  MoveL 7398 to (239.35, 44.42, 106.87) mm, rotated rx -180 ry 0 rz 180 deg; joints [-29.24, 54.738, -85.05, 32.961, 116.129, 15.937]
  Call Extruder(207.44470)
  MoveL 7399 to (239.44, 44.66, 106.87) mm, rotated rx 180 ry 0 rz 180 deg; joints [-29.343, 54.76, -85.048, 33.066, 116.082, 15.973]
  MoveL 7400 to (239.44, 44.66, 106.87) mm, rotated rx 180 ry 0 rz 180 deg; joints [-29.343, 54.76, -85.048, 33.066, 116.082, 15.973]
  Call Extruder(207.55794)
  MoveL 7401 to (239.5, 44.85, 106.87) mm, rotated rx 180 ry 0 rz 180 deg; joints [-29.428, 54.775, -85.047, 33.152, 116.044, 16.002]
  MoveL 7402 to (239.5, 44.85, 106.87) mm, rotated rx 180 ry 0 rz 180 deg; joints [-29.428, 54.775, -85.047, 33.152, 116.044, 16.002]
  Call Extruder(207.67073)
  MoveL 7403 to (239.56, 45.03, 106.87) mm, rotated rx 180 ry 0 rz 180 deg; joints [-29.512, 54.791, -85.047, 33.237, 116.007, 16.031]
  MoveL 7404 to (239.56, 45.03, 106.87) mm, rotated rx 180 ry 0 rz 180 deg; joints [-29.512, 54.791, -85.047, 33.237, 116.007, 16.031]
  Call Extruder(207.78308)
  MoveL 7405 to (239.62, 45.22, 106.87) mm, rotated rx -180 ry 0 rz 180 deg; joints [-29.596, 54.807, -85.046, 33.322, 115.97, 16.061]
  MoveL 7406 to (239.62, 45.22, 106.87) mm, rotated rx -180 ry 0 rz 180 deg; joints [-29.596, 54.807, -85.046, 33.322, 115.97, 16.061]
  Call Extruder(207.89498)
  MoveL 7407 to (239.68, 45.41, 106.87) mm, rotated rx 180 ry 0 rz 180 deg; joints [-29.679, 54.822, -85.045, 33.407, 115.933, 16.089]
  MoveL 7408 to (239.68, 45.41, 106.87) mm, rotated rx 180 ry 0 rz 180 deg; joints [-29.679, 54.822, -85.045, 33.407, 115.933, 16.089]
  Call Extruder(208.01638)
  MoveL 7409 to (239.75, 45.62, 106.87) mm, rotated rx -180 ry 0 rz 180 deg; joints [-29.77, 54.839, -85.044, 33.5, 115.893, 16.121]
  MoveL 7410 to (239.75, 45.62, 106.87) mm, rotated rx -180 ry 0 rz 180 deg; joints [-29.77, 54.839, -85.044, 33.5, 115.893, 16.121]
  Call Extruder(208.14717)
  MoveL 7411 to (239.82, 45.84, 106.87) mm, rotated rx 180 ry 0 rz -180 deg; joints [-29.871, 54.858, -85.043, 33.601, 115.849, 16.156]
  MoveL 7412 to (239.82, 45.84, 106.87) mm, rotated rx 180 ry 0 rz -180 deg; joints [-29.871, 54.858, -85.043, 33.601, 115.849, 16.156]
  Call Extruder(208.27740)
  MoveL 7413 to (239.88, 46.06, 106.87) mm, rotated rx -180 ry 0 rz 180 deg; joints [-29.97, 54.876, -85.041, 33.702, 115.805, 16.19]
  MoveL 7414 to (239.88, 46.06, 106.87) mm, rotated rx -180 ry 0 rz 180 deg; joints [-29.97, 54.876, -85.041, 33.702, 115.805, 16.19]
  Call Extruder(208.40706)
  MoveL 7415 to (239.95, 46.29, 106.87) mm, rotated rx -180 ry 0 rz 180 deg; joints [-30.069, 54.894, -85.04, 33.803, 115.761, 16.224]
  MoveL 7416 to (239.95, 46.29, 106.87) mm, rotated rx -180 ry 0 rz 180 deg; joints [-30.069, 54.894, -85.04, 33.803, 115.761, 16.224]
  Call Extruder(208.53615)
  MoveL 7417 to (240.02, 46.51, 106.87) mm, rotated rx -180 ry 0 rz 180 deg; joints [-30.168, 54.913, -85.039, 33.903, 115.717, 16.258]
  MoveL 7418 to (240.02, 46.51, 106.87) mm, rotated rx -180 ry 0 rz 180 deg; joints [-30.168, 54.913, -85.039, 33.903, 115.717, 16.258]
  Call Extruder(208.65121)
  MoveL 7419 to (240.06, 46.72, 106.87) mm, rotated rx 180 ry 0 rz 180 deg; joints [-30.263, 54.928, -85.038, 34, 115.677, 16.292]
  MoveL 7420 to (240.06, 46.72, 106.87) mm, rotated rx 180 ry 0 rz 180 deg; joints [-30.263, 54.928, -85.038, 34, 115.677, 16.292]
  Call Extruder(208.76581)
  MoveL 7421 to (240.11, 46.92, 106.87) mm, rotated rx -180 ry 0 rz 180 deg; joints [-30.358, 54.943, -85.037, 34.097, 115.637, 16.326]
  MoveL 7422 to (240.11, 46.92, 106.87) mm, rotated rx -180 ry 0 rz 180 deg; joints [-30.358, 54.943, -85.037, 34.097, 115.637, 16.326]
  Call Extruder(208.87996)
  MoveL 7423 to (240.15, 47.12, 106.87) mm, rotated rx -180 ry 0 rz 180 deg; joints [-30.453, 54.958, -85.036, 34.193, 115.597, 16.359]
  MoveL 7424 to (240.15, 47.12, 106.87) mm, rotated rx -180 ry 0 rz 180 deg; joints [-30.453, 54.958, -85.036, 34.193, 115.597, 16.359]
  Call Extruder(208.99365)
  MoveL 7425 to (240.2, 47.33, 106.87) mm, rotated rx 180 ry 0 rz 180 deg; joints [-30.548, 54.973, -85.035, 34.29, 115.557, 16.393]
  MoveL 7426 to (240.2, 47.33, 106.87) mm, rotated rx 180 ry 0 rz 180 deg; joints [-30.548, 54.973, -85.035, 34.29, 115.557, 16.393]
  Call Extruder(209.11906)
  MoveL 7427 to (240.24, 47.55, 106.87) mm, rotated rx -180 ry 0 rz 180 deg; joints [-30.653, 54.99, -85.034, 34.396, 115.513, 16.43]
  MoveL 7428 to (240.24, 47.55, 106.87) mm, rotated rx -180 ry 0 rz 180 deg; joints [-30.653, 54.99, -85.034, 34.396, 115.513, 16.43]
  Call Extruder(209.25604)
  MoveL 7429 to (240.29, 47.8, 106.87) mm, rotated rx 180 ry 0 rz -180 deg; joints [-30.768, 55.008, -85.033, 34.514, 115.464, 16.47]
  MoveL 7430 to (240.29, 47.8, 106.87) mm, rotated rx 180 ry 0 rz -180 deg; joints [-30.768, 55.008, -85.033, 34.514, 115.464, 16.47]
  Call Extruder(209.39241)
  MoveL 7431 to (240.34, 48.05, 106.87) mm, rotated rx -180 ry 0 rz 180 deg; joints [-30.884, 55.026, -85.032, 34.632, 115.415, 16.511]
  MoveL 7432 to (240.34, 48.05, 106.87) mm, rotated rx -180 ry 0 rz 180 deg; joints [-30.884, 55.026, -85.032, 34.632, 115.415, 16.511]
  Call Extruder(209.52817)
  MoveL 7433 to (240.39, 48.3, 106.87) mm, rotated rx -180 ry 0 rz 180 deg; joints [-30.999, 55.045, -85.031, 34.749, 115.366, 16.551]
  MoveL 7434 to (240.39, 48.3, 106.87) mm, rotated rx -180 ry 0 rz 180 deg; joints [-30.999, 55.045, -85.031, 34.749, 115.366, 16.551]
  Call Extruder(209.66331)
  MoveL 7435 to (240.44, 48.55, 106.87) mm, rotated rx 180 ry 0 rz 180 deg; joints [-31.114, 55.063, -85.029, 34.865, 115.318, 16.591]
  MoveL 7436 to (240.44, 48.55, 106.87) mm, rotated rx 180 ry 0 rz 180 deg; joints [-31.114, 55.063, -85.029, 34.865, 115.318, 16.591]
  Call Extruder(209.79785)
  MoveL 7437 to (240.49, 48.8, 106.87) mm, rotated rx -180 ry 0 rz 180 deg; joints [-31.228, 55.081, -85.028, 34.981, 115.269, 16.63]
  MoveL 7438 to (240.49, 48.8, 106.87) mm, rotated rx -180 ry 0 rz 180 deg; joints [-31.228, 55.081, -85.028, 34.981, 115.269, 16.63]
  Call Extruder(209.93178)
  MoveL 7439 to (240.54, 49.05, 106.87) mm, rotated rx -180 ry 0 rz 180 deg; joints [-31.342, 55.1, -85.027, 35.096, 115.22, 16.669]
  MoveL 7440 to (240.54, 49.05, 106.87) mm, rotated rx -180 ry 0 rz 180 deg; joints [-31.342, 55.1, -85.027, 35.096, 115.22, 16.669]
  Call Extruder(210.07964)
  MoveL 7441 to (240.59, 49.33, 106.87) mm, rotated rx -180 ry 0 rz 180 deg; joints [-31.47, 55.12, -85.026, 35.226, 115.166, 16.713]
  MoveL 7442 to (240.59, 49.33, 106.87) mm, rotated rx -180 ry 0 rz 180 deg; joints [-31.47, 55.12, -85.026, 35.226, 115.166, 16.713]
  Call Extruder(210.24139)
  MoveL 7443 to (240.64, 49.63, 106.87) mm, rotated rx -180 ry 0 rz 180 deg; joints [-31.612, 55.141, -85.024, 35.37, 115.106, 16.762]
  MoveL 7444 to (240.64, 49.63, 106.87) mm, rotated rx -180 ry 0 rz 180 deg; joints [-31.612, 55.141, -85.024, 35.37, 115.106, 16.762]
  Call Extruder(210.40241)
  MoveL 7445 to (240.69, 49.94, 106.87) mm, rotated rx -180 ry 0 rz 180 deg; joints [-31.755, 55.163, -85.023, 35.514, 115.046, 16.811]
  MoveL 7446 to (240.69, 49.94, 106.87) mm, rotated rx -180 ry 0 rz 180 deg; joints [-31.755, 55.163, -85.023, 35.514, 115.046, 16.811]
  Call Extruder(210.56270)
  MoveL 7447 to (240.74, 50.24, 106.87) mm, rotated rx -180 ry 0 rz 180 deg; joints [-31.895, 55.184, -85.021, 35.657, 114.987, 16.859]
  MoveL 7448 to (240.74, 50.24, 106.87) mm, rotated rx -180 ry 0 rz 180 deg; joints [-31.895, 55.184, -85.021, 35.657, 114.987, 16.859]
  Call Extruder(210.72226)
  MoveL 7449 to (240.78, 50.55, 106.87) mm, rotated rx 180 ry 0 rz 180 deg; joints [-32.036, 55.206, -85.019, 35.799, 114.927, 16.907]
  MoveL 7450 to (240.78, 50.55, 106.87) mm, rotated rx 180 ry 0 rz 180 deg; joints [-32.036, 55.206, -85.019, 35.799, 114.927, 16.907]
  Call Extruder(210.88109)
  MoveL 7451 to (240.83, 50.86, 106.87) mm, rotated rx -180 ry 0 rz 180 deg; joints [-32.176, 55.228, -85.018, 35.941, 114.867, 16.954]
  MoveL 7452 to (240.83, 50.86, 106.87) mm, rotated rx -180 ry 0 rz 180 deg; joints [-32.176, 55.228, -85.018, 35.941, 114.867, 16.954]
  Call Extruder(211.05976)
  MoveL 7453 to (240.88, 51.2, 106.87) mm, rotated rx -180 ry 0 rz 180 deg; joints [-32.337, 55.252, -85.016, 36.103, 114.8, 17.009]
  MoveL 7454 to (240.88, 51.2, 106.87) mm, rotated rx -180 ry 0 rz 180 deg; joints [-32.337, 55.252, -85.016, 36.103, 114.8, 17.009]
  Call Extruder(211.25821)
  MoveL 7455 to (240.93, 51.59, 106.87) mm, rotated rx -180 ry 0 rz 180 deg; joints [-32.518, 55.278, -85.014, 36.285, 114.724, 17.07]
  MoveL 7456 to (240.93, 51.59, 106.87) mm, rotated rx -180 ry 0 rz 180 deg; joints [-32.518, 55.278, -85.014, 36.285, 114.724, 17.07]
  Call Extruder(211.45578)
  MoveL 7457 to (240.97, 51.98, 106.87) mm, rotated rx 180 ry 0 rz 180 deg; joints [-32.697, 55.304, -85.012, 36.467, 114.648, 17.131]
  MoveL 7458 to (240.97, 51.98, 106.87) mm, rotated rx 180 ry 0 rz 180 deg; joints [-32.697, 55.304, -85.012, 36.467, 114.648, 17.131]
  Call Extruder(211.65249)
  MoveL 7459 to (241.02, 52.37, 106.87) mm, rotated rx -180 ry 0 rz 180 deg; joints [-32.876, 55.331, -85.01, 36.647, 114.573, 17.19]
  MoveL 7460 to (241.02, 52.37, 106.87) mm, rotated rx -180 ry 0 rz 180 deg; joints [-32.876, 55.331, -85.01, 36.647, 114.573, 17.19]
  Call Extruder(211.84833)
  MoveL 7461 to (241.06, 52.75, 106.87) mm, rotated rx -180 ry 0 rz 180 deg; joints [-33.055, 55.357, -85.008, 36.826, 114.497, 17.249]
  MoveL 7462 to (241.06, 52.75, 106.87) mm, rotated rx -180 ry 0 rz 180 deg; joints [-33.055, 55.357, -85.008, 36.826, 114.497, 17.249]
  Call Extruder(212.14376)
  MoveL 7463 to (241.11, 53.34, 106.87) mm, rotated rx 180 ry 0 rz 180 deg; joints [-33.331, 55.396, -85.005, 37.105, 114.382, 17.342]
  MoveL 7464 to (241.11, 53.34, 106.87) mm, rotated rx 180 ry 0 rz 180 deg; joints [-33.331, 55.396, -85.005, 37.105, 114.382, 17.342]
  Call Extruder(212.43787)
  MoveL 7465 to (241.15, 53.93, 106.87) mm, rotated rx -180 ry 0 rz 180 deg; joints [-33.606, 55.434, -85.002, 37.381, 114.266, 17.433]
  MoveL 7466 to (241.15, 53.93, 106.87) mm, rotated rx -180 ry 0 rz 180 deg; joints [-33.606, 55.434, -85.002, 37.381, 114.266, 17.433]
  Call Extruder(212.73064)
  MoveL 7467 to (241.2, 54.52, 106.87) mm, rotated rx 180 ry 0 rz 180 deg; joints [-33.878, 55.473, -84.999, 37.655, 114.151, 17.521]
  MoveL 7468 to (241.2, 54.52, 106.87) mm, rotated rx 180 ry 0 rz 180 deg; joints [-33.878, 55.473, -84.999, 37.655, 114.151, 17.521]
  Call Extruder(213.30409)
  MoveL 7469 to (241.25, 55.68, 106.87) mm, rotated rx -180 ry 0 rz 180 deg; joints [-34.425, 55.546, -84.993, 38.203, 113.923, 17.7]
  MoveL 7470 to (241.25, 55.68, 106.87) mm, rotated rx -180 ry 0 rz 180 deg; joints [-34.425, 55.546, -84.993, 38.203, 113.923, 17.7]
  Call Extruder(214.01793)
  MoveL 7471 to (241.29, 57.14, 106.87) mm, rotated rx -180 ry 0 rz 180 deg; joints [-35.104, 55.637, -84.985, 38.883, 113.638, 17.918]
  Call Extruder(256.08281)
  MoveL 7472 to (241.29, 142.86, 106.87) mm, rotated rx 180 ry 0 rz 180 deg; joints [-60.361, 61.969, -83.576, 62.121, 100.493, 18.996]
  Call Extruder(256.51124)
  MoveL 7473 to (241.27, 143.74, 106.87) mm, rotated rx 180 ry 0 rz 180 deg; joints [-60.516, 62.035, -83.55, 62.255, 100.399, 18.94]
  MoveL 7474 to (241.27, 143.74, 106.87) mm, rotated rx 180 ry 0 rz 180 deg; joints [-60.516, 62.035, -83.55, 62.255, 100.399, 18.94]
  Call Extruder(257.08469)
  MoveL 7475 to (241.23, 144.9, 106.87) mm, rotated rx -180 ry 0 rz 180 deg; joints [-60.726, 62.123, -83.516, 62.438, 100.275, 18.867]
  MoveL 7476 to (241.23, 144.9, 106.87) mm, rotated rx -180 ry 0 rz 180 deg; joints [-60.726, 62.123, -83.516, 62.438, 100.275, 18.867]
  Call Extruder(257.51903)
  MoveL 7477 to (241.18, 145.77, 106.87) mm, rotated rx -180 ry 0 rz 180 deg; joints [-60.887, 62.188, -83.49, 62.578, 100.181, 18.812]
  MoveL 7478 to (241.18, 145.77, 106.87) mm, rotated rx -180 ry 0 rz 180 deg; joints [-60.887, 62.188, -83.49, 62.578, 100.181, 18.812]
  Call Extruder(257.81314)
  MoveL 7479 to (241.13, 146.36, 106.87) mm, rotated rx -180 ry 0 rz 180 deg; joints [-61, 62.231, -83.473, 62.676, 100.117, 18.777]
  MoveL 7480 to (241.13, 146.36, 106.87) mm, rotated rx -180 ry 0 rz 180 deg; joints [-61, 62.231, -83.473, 62.676, 100.117, 18.777]
  Call Extruder(258.10858)
  MoveL 7481 to (241.09, 146.95, 106.87) mm, rotated rx -180 ry 0 rz 180 deg; joints [-61.111, 62.275, -83.456, 62.774, 100.053, 18.741]
  MoveL 7482 to (241.09, 146.95, 106.87) mm, rotated rx -180 ry 0 rz 180 deg; joints [-61.111, 62.275, -83.456, 62.774, 100.053, 18.741]
  Call Extruder(258.35483)
  MoveL 7483 to (241.04, 147.44, 106.87) mm, rotated rx 180 ry 0 rz -180 deg; joints [-61.205, 62.31, -83.441, 62.857, 100, 18.712]
  MoveL 7484 to (241.04, 147.44, 106.87) mm, rotated rx 180 ry 0 rz -180 deg; joints [-61.205, 62.31, -83.441, 62.857, 100, 18.712]
  Call Extruder(258.55154)
  MoveL 7485 to (240.99, 147.83, 106.87) mm, rotated rx -180 ry 0 rz 180 deg; joints [-61.282, 62.338, -83.43, 62.925, 99.957, 18.689]
  MoveL 7486 to (240.99, 147.83, 106.87) mm, rotated rx -180 ry 0 rz 180 deg; joints [-61.282, 62.338, -83.43, 62.925, 99.957, 18.689]
  Call Extruder(258.74911)
  MoveL 7487 to (240.95, 148.22, 106.87) mm, rotated rx -180 ry 0 rz 180 deg; joints [-61.359, 62.366, -83.419, 62.992, 99.915, 18.667]
  MoveL 7488 to (240.95, 148.22, 106.87) mm, rotated rx -180 ry 0 rz 180 deg; joints [-61.359, 62.366, -83.419, 62.992, 99.915, 18.667]
  Call Extruder(258.94755)
  MoveL 7489 to (240.9, 148.6, 106.87) mm, rotated rx 180 ry 0 rz -180 deg; joints [-61.436, 62.393, -83.407, 63.06, 99.873, 18.644]
  MoveL 7490 to (240.9, 148.6, 106.87) mm, rotated rx 180 ry 0 rz -180 deg; joints [-61.436, 62.393, -83.407, 63.06, 99.873, 18.644]
  Call Extruder(259.14686)
  MoveL 7491 to (240.86, 148.99, 106.87) mm, rotated rx -180 ry 0 rz 180 deg; joints [-61.512, 62.421, -83.396, 63.127, 99.831, 18.621]
  MoveL 7492 to (240.86, 148.99, 106.87) mm, rotated rx -180 ry 0 rz 180 deg; joints [-61.512, 62.421, -83.396, 63.127, 99.831, 18.621]
  Call Extruder(259.30569)
  MoveL 7493 to (240.81, 149.3, 106.87) mm, rotated rx -180 ry 0 rz -180 deg; joints [-61.575, 62.443, -83.387, 63.184, 99.797, 18.604]
  MoveL 7494 to (240.81, 149.3, 106.87) mm, rotated rx -180 ry 0 rz -180 deg; joints [-61.575, 62.443, -83.387, 63.184, 99.797, 18.604]
  Call Extruder(259.46525)
  MoveL 7495 to (240.76, 149.6, 106.87) mm, rotated rx 180 ry 0 rz 180 deg; joints [-61.639, 62.464, -83.378, 63.24, 99.763, 18.587]
  MoveL 7496 to (240.76, 149.6, 106.87) mm, rotated rx 180 ry 0 rz 180 deg; joints [-61.639, 62.464, -83.378, 63.24, 99.763, 18.587]
  Call Extruder(259.62554)
  MoveL 7497 to (240.71, 149.91, 106.87) mm, rotated rx 180 ry 0 rz 180 deg; joints [-61.702, 62.485, -83.369, 63.296, 99.729, 18.57]
  MoveL 7498 to (240.71, 149.91, 106.87) mm, rotated rx 180 ry 0 rz 180 deg; joints [-61.702, 62.485, -83.369, 63.296, 99.729, 18.57]
  Call Extruder(259.78655)
  MoveL 7499 to (240.66, 150.21, 106.87) mm, rotated rx 180 ry 0 rz 180 deg; joints [-61.765, 62.507, -83.36, 63.352, 99.695, 18.552]
  MoveL 7500 to (240.66, 150.21, 106.87) mm, rotated rx 180 ry 0 rz 180 deg; joints [-61.765, 62.507, -83.36, 63.352, 99.695, 18.552]
  Call Extruder(259.94830)
  MoveL 7501 to (240.61, 150.52, 106.87) mm, rotated rx -180 ry 0 rz 180 deg; joints [-61.828, 62.528, -83.351, 63.408, 99.662, 18.535]
  MoveL 7502 to (240.61, 150.52, 106.87) mm, rotated rx -180 ry 0 rz 180 deg; joints [-61.828, 62.528, -83.351, 63.408, 99.662, 18.535]
  Call Extruder(260.11077)
  MoveL 7503 to (240.56, 150.83, 106.87) mm, rotated rx 180 ry 0 rz 180 deg; joints [-61.891, 62.55, -83.342, 63.464, 99.628, 18.518]
  MoveL 7504 to (240.56, 150.83, 106.87) mm, rotated rx 180 ry 0 rz 180 deg; joints [-61.891, 62.55, -83.342, 63.464, 99.628, 18.518]
  Call Extruder(260.24469)
  MoveL 7505 to (240.52, 151.07, 106.87) mm, rotated rx 180 ry 0 rz 180 deg; joints [-61.944, 62.567, -83.335, 63.512, 99.6, 18.504]
  MoveL 7506 to (240.52, 151.07, 106.87) mm, rotated rx 180 ry 0 rz 180 deg; joints [-61.944, 62.567, -83.335, 63.512, 99.6, 18.504]
  Call Extruder(260.37923)
  MoveL 7507 to (240.47, 151.32, 106.87) mm, rotated rx -180 ry 0 rz 180 deg; joints [-61.998, 62.584, -83.328, 63.56, 99.573, 18.491]
  MoveL 7508 to (240.47, 151.32, 106.87) mm, rotated rx -180 ry 0 rz 180 deg; joints [-61.998, 62.584, -83.328, 63.56, 99.573, 18.491]
  Call Extruder(260.51438)
  MoveL 7509 to (240.42, 151.57, 106.87) mm, rotated rx -180 ry 0 rz 180 deg; joints [-62.052, 62.601, -83.321, 63.608, 99.545, 18.477]
  MoveL 7510 to (240.42, 151.57, 106.87) mm, rotated rx -180 ry 0 rz 180 deg; joints [-62.052, 62.601, -83.321, 63.608, 99.545, 18.477]
  Call Extruder(260.65014)
  MoveL 7511 to (240.37, 151.82, 106.87) mm, rotated rx 180 ry 0 rz 180 deg; joints [-62.105, 62.618, -83.314, 63.656, 99.517, 18.464]
  MoveL 7512 to (240.37, 151.82, 106.87) mm, rotated rx 180 ry 0 rz 180 deg; joints [-62.105, 62.618, -83.314, 63.656, 99.517, 18.464]
  Call Extruder(260.78650)
  MoveL 7513 to (240.32, 152.07, 106.87) mm, rotated rx -180 ry 0 rz -180 deg; joints [-62.159, 62.635, -83.306, 63.704, 99.489, 18.45]
  MoveL 7514 to (240.32, 152.07, 106.87) mm, rotated rx -180 ry 0 rz -180 deg; joints [-62.159, 62.635, -83.306, 63.704, 99.489, 18.45]
  Call Extruder(260.92348)
  MoveL 7515 to (240.27, 152.32, 106.87) mm, rotated rx 180 ry 0 rz -180 deg; joints [-62.212, 62.652, -83.299, 63.751, 99.462, 18.437]
  MoveL 7516 to (240.27, 152.32, 106.87) mm, rotated rx 180 ry 0 rz -180 deg; joints [-62.212, 62.652, -83.299, 63.751, 99.462, 18.437]
  Call Extruder(261.06107)
  MoveL 7517 to (240.22, 152.57, 106.87) mm, rotated rx -180 ry 0 rz 180 deg; joints [-62.265, 62.669, -83.292, 63.799, 99.434, 18.423]
  MoveL 7518 to (240.22, 152.57, 106.87) mm, rotated rx -180 ry 0 rz 180 deg; joints [-62.265, 62.669, -83.292, 63.799, 99.434, 18.423]
  Call Extruder(261.17477)
  MoveL 7519 to (240.17, 152.77, 106.87) mm, rotated rx -180 ry 0 rz 180 deg; joints [-62.31, 62.683, -83.286, 63.839, 99.411, 18.412]
  MoveL 7520 to (240.17, 152.77, 106.87) mm, rotated rx -180 ry 0 rz 180 deg; joints [-62.31, 62.683, -83.286, 63.839, 99.411, 18.412]
  Call Extruder(261.28892)
  MoveL 7521 to (240.13, 152.98, 106.87) mm, rotated rx -180 ry 0 rz 180 deg; joints [-62.355, 62.696, -83.28, 63.879, 99.389, 18.401]
  MoveL 7522 to (240.13, 152.98, 106.87) mm, rotated rx -180 ry 0 rz 180 deg; joints [-62.355, 62.696, -83.28, 63.879, 99.389, 18.401]
  Call Extruder(261.40352)
  MoveL 7523 to (240.08, 153.18, 106.87) mm, rotated rx -180 ry 0 rz 180 deg; joints [-62.399, 62.71, -83.274, 63.919, 99.366, 18.39]
  MoveL 7524 to (240.08, 153.18, 106.87) mm, rotated rx -180 ry 0 rz 180 deg; joints [-62.399, 62.71, -83.274, 63.919, 99.366, 18.39]
  Call Extruder(261.51858)
  MoveL 7525 to (240.04, 153.39, 106.87) mm, rotated rx 180 ry 0 rz 180 deg; joints [-62.444, 62.724, -83.268, 63.958, 99.343, 18.379]
  MoveL 7526 to (240.04, 153.39, 106.87) mm, rotated rx 180 ry 0 rz 180 deg; joints [-62.444, 62.724, -83.268, 63.958, 99.343, 18.379]
  Call Extruder(261.64080)
  MoveL 7527 to (239.98, 153.6, 106.87) mm, rotated rx 180 ry 0 rz 180 deg; joints [-62.493, 62.738, -83.262, 64.003, 99.319, 18.368]
  MoveL 7528 to (239.98, 153.6, 106.87) mm, rotated rx 180 ry 0 rz 180 deg; joints [-62.493, 62.738, -83.262, 64.003, 99.319, 18.368]
  Call Extruder(261.77046)
  MoveL 7529 to (239.92, 153.82, 106.87) mm, rotated rx 180 ry 0 rz -180 deg; joints [-62.547, 62.752, -83.256, 64.052, 99.293, 18.358]
  MoveL 7530 to (239.92, 153.82, 106.87) mm, rotated rx 180 ry 0 rz -180 deg; joints [-62.547, 62.752, -83.256, 64.052, 99.293, 18.358]
  Call Extruder(261.90069)
  MoveL 7531 to (239.85, 154.05, 106.87) mm, rotated rx 180 ry 0 rz 180 deg; joints [-62.601, 62.767, -83.249, 64.1, 99.267, 18.347]
  MoveL 7532 to (239.85, 154.05, 106.87) mm, rotated rx 180 ry 0 rz 180 deg; joints [-62.601, 62.767, -83.249, 64.1, 99.267, 18.347]
  Call Extruder(262.03148)
  MoveL 7533 to (239.78, 154.27, 106.87) mm, rotated rx -180 ry 0 rz 180 deg; joints [-62.654, 62.781, -83.243, 64.149, 99.241, 18.337]
  MoveL 7534 to (239.78, 154.27, 106.87) mm, rotated rx -180 ry 0 rz 180 deg; joints [-62.654, 62.781, -83.243, 64.149, 99.241, 18.337]
  Call Extruder(262.16284)
  MoveL 7535 to (239.71, 154.49, 106.87) mm, rotated rx 180 ry 0 rz 180 deg; joints [-62.708, 62.796, -83.237, 64.198, 99.215, 18.326]
  MoveL 7536 to (239.71, 154.49, 106.87) mm, rotated rx 180 ry 0 rz 180 deg; joints [-62.708, 62.796, -83.237, 64.198, 99.215, 18.326]
  Call Extruder(262.27474)
  MoveL 7537 to (239.65, 154.68, 106.87) mm, rotated rx 180 ry 0 rz 180 deg; joints [-62.754, 62.808, -83.232, 64.24, 99.193, 18.318]
  MoveL 7538 to (239.65, 154.68, 106.87) mm, rotated rx 180 ry 0 rz 180 deg; joints [-62.754, 62.808, -83.232, 64.24, 99.193, 18.318]
  Call Extruder(262.38708)
  MoveL 7539 to (239.59, 154.87, 106.87) mm, rotated rx 180 ry 0 rz 180 deg; joints [-62.801, 62.82, -83.226, 64.282, 99.171, 18.309]
  MoveL 7540 to (239.59, 154.87, 106.87) mm, rotated rx 180 ry 0 rz 180 deg; joints [-62.801, 62.82, -83.226, 64.282, 99.171, 18.309]
  Call Extruder(262.49987)
  MoveL 7541 to (239.53, 155.06, 106.87) mm, rotated rx 180 ry 0 rz 180 deg; joints [-62.847, 62.832, -83.221, 64.324, 99.149, 18.3]
  MoveL 7542 to (239.53, 155.06, 106.87) mm, rotated rx 180 ry 0 rz 180 deg; joints [-62.847, 62.832, -83.221, 64.324, 99.149, 18.3]
  Call Extruder(262.61311)
  MoveL 7543 to (239.47, 155.25, 106.87) mm, rotated rx -180 ry 0 rz 180 deg; joints [-62.893, 62.844, -83.216, 64.366, 99.127, 18.292]
  MoveL 7544 to (239.47, 155.25, 106.87) mm, rotated rx -180 ry 0 rz 180 deg; joints [-62.893, 62.844, -83.216, 64.366, 99.127, 18.292]
  Call Extruder(262.72679)
  MoveL 7545 to (239.41, 155.44, 106.87) mm, rotated rx 180 ry 0 rz -180 deg; joints [-62.939, 62.856, -83.21, 64.407, 99.105, 18.283]
  MoveL 7546 to (239.41, 155.44, 106.87) mm, rotated rx 180 ry 0 rz -180 deg; joints [-62.939, 62.856, -83.21, 64.407, 99.105, 18.283]
  Call Extruder(262.90875)
  MoveL 7547 to (239.29, 155.73, 106.87) mm, rotated rx 180 ry 0 rz 180 deg; joints [-63.018, 62.873, -83.203, 64.48, 99.069, 18.272]
  MoveL 7548 to (239.29, 155.73, 106.87) mm, rotated rx 180 ry 0 rz 180 deg; joints [-63.018, 62.873, -83.203, 64.48, 99.069, 18.272]
  Call Extruder(263.09146)
  MoveL 7549 to (239.16, 156.02, 106.87) mm, rotated rx 180 ry 0 rz 180 deg; joints [-63.097, 62.891, -83.195, 64.552, 99.034, 18.26]
  MoveL 7550 to (239.16, 156.02, 106.87) mm, rotated rx 180 ry 0 rz 180 deg; joints [-63.097, 62.891, -83.195, 64.552, 99.034, 18.26]
  Call Extruder(263.26189)
  MoveL 7551 to (239.05, 156.29, 106.87) mm, rotated rx -180 ry 0 rz 180 deg; joints [-63.17, 62.907, -83.188, 64.619, 99.001, 18.25]
  MoveL 7552 to (239.05, 156.29, 106.87) mm, rotated rx -180 ry 0 rz 180 deg; joints [-63.17, 62.907, -83.188, 64.619, 99.001, 18.25]
  Call Extruder(263.41990)
  MoveL 7553 to (238.94, 156.54, 106.87) mm, rotated rx 180 ry 0 rz 180 deg; joints [-63.238, 62.922, -83.181, 64.681, 98.97, 18.241]
  MoveL 7554 to (238.94, 156.54, 106.87) mm, rotated rx 180 ry 0 rz 180 deg; joints [-63.238, 62.922, -83.181, 64.681, 98.97, 18.241]
  Call Extruder(263.57851)
  MoveL 7555 to (238.84, 156.79, 106.87) mm, rotated rx 180 ry 0 rz 180 deg; joints [-63.306, 62.937, -83.174, 64.743, 98.94, 18.231]
  MoveL 7556 to (238.84, 156.79, 106.87) mm, rotated rx 180 ry 0 rz 180 deg; joints [-63.306, 62.937, -83.174, 64.743, 98.94, 18.231]
  Call Extruder(263.78468)
  MoveL 7557 to (238.66, 157.09, 106.87) mm, rotated rx 180 ry 0 rz 180 deg; joints [-63.401, 62.953, -83.167, 64.832, 98.9, 18.223]
  MoveL 7558 to (238.66, 157.09, 106.87) mm, rotated rx 180 ry 0 rz 180 deg; joints [-63.401, 62.953, -83.167, 64.832, 98.9, 18.223]
  Call Extruder(263.99163)
  MoveL 7559 to (238.49, 157.4, 106.87) mm, rotated rx -180 ry 0 rz -180 deg; joints [-63.497, 62.97, -83.16, 64.92, 98.86, 18.216]
  MoveL 7560 to (238.49, 157.4, 106.87) mm, rotated rx -180 ry 0 rz -180 deg; joints [-63.497, 62.97, -83.16, 64.92, 98.86, 18.216]
  Call Extruder(264.19935)
  MoveL 7561 to (238.31, 157.7, 106.87) mm, rotated rx -180 ry 0 rz -180 deg; joints [-63.592, 62.986, -83.152, 65.008, 98.82, 18.208]
  MoveL 7562 to (238.31, 157.7, 106.87) mm, rotated rx -180 ry 0 rz -180 deg; joints [-63.592, 62.986, -83.152, 65.008, 98.82, 18.208]
  Call Extruder(264.40786)
  MoveL 7563 to (238.14, 158.01, 106.87) mm, rotated rx -180 ry 0 rz 180 deg; joints [-63.687, 63.003, -83.145, 65.096, 98.78, 18.2]
  MoveL 7564 to (238.14, 158.01, 106.87) mm, rotated rx -180 ry 0 rz 180 deg; joints [-63.687, 63.003, -83.145, 65.096, 98.78, 18.2]
  Call Extruder(264.58740)
  MoveL 7565 to (237.96, 158.25, 106.87) mm, rotated rx -180 ry 0 rz 180 deg; joints [-63.774, 63.015, -83.139, 65.177, 98.745, 18.196]
  MoveL 7566 to (237.96, 158.25, 106.87) mm, rotated rx -180 ry 0 rz 180 deg; joints [-63.774, 63.015, -83.139, 65.177, 98.745, 18.196]
  Call Extruder(264.92080)
  MoveL 7567 to (237.63, 158.7, 106.87) mm, rotated rx -180 ry 0 rz 180 deg; joints [-63.934, 63.037, -83.129, 65.326, 98.682, 18.19]
  MoveL 7568 to (237.63, 158.7, 106.87) mm, rotated rx -180 ry 0 rz 180 deg; joints [-63.934, 63.037, -83.129, 65.326, 98.682, 18.19]
  Call Extruder(265.25540)
  MoveL 7569 to (237.3, 159.15, 106.87) mm, rotated rx 180 ry 0 rz 180 deg; joints [-64.094, 63.059, -83.119, 65.475, 98.619, 18.183]
  Call Extruder(266.08335)
  MoveL 7570 to (236.39, 160.19, 106.87) mm, rotated rx -180 ry 0 rz 180 deg; joints [-64.505, 63.105, -83.098, 65.861, 98.463, 18.18]
  Call Extruder(266.91129)
  MoveL 7571 to (235.35, 161.1, 106.87) mm, rotated rx -180 ry 0 rz -180 deg; joints [-64.933, 63.137, -83.083, 66.266, 98.31, 18.197]
  Call Extruder(267.07860)
  MoveL 7572 to (235.13, 161.27, 106.87) mm, rotated rx -180 ry 0 rz 180 deg; joints [-65.021, 63.142, -83.081, 66.35, 98.28, 18.203]
  MoveL 7573 to (235.13, 161.27, 106.87) mm, rotated rx -180 ry 0 rz 180 deg; joints [-65.021, 63.142, -83.081, 66.35, 98.28, 18.203]
  Call Extruder(267.41202)
  MoveL 7574 to (234.68, 161.59, 106.87) mm, rotated rx 180 ry 0 rz 180 deg; joints [-65.197, 63.151, -83.077, 66.517, 98.219, 18.215]
  MoveL 7575 to (234.68, 161.59, 106.87) mm, rotated rx 180 ry 0 rz 180 deg; joints [-65.197, 63.151, -83.077, 66.517, 98.219, 18.215]
  Call Extruder(267.74426)
  MoveL 7576 to (234.23, 161.92, 106.87) mm, rotated rx 180 ry 0 rz 180 deg; joints [-65.374, 63.16, -83.073, 66.684, 98.159, 18.226]
  MoveL 7577 to (234.23, 161.92, 106.87) mm, rotated rx 180 ry 0 rz 180 deg; joints [-65.374, 63.16, -83.073, 66.684, 98.159, 18.226]
  Call Extruder(267.86192)
  MoveL 7578 to (234.05, 162.02, 106.87) mm, rotated rx 180 ry 0 rz -180 deg; joints [-65.437, 63.162, -83.072, 66.745, 98.138, 18.233]
  MoveL 7579 to (234.05, 162.02, 106.87) mm, rotated rx 180 ry 0 rz -180 deg; joints [-65.437, 63.162, -83.072, 66.745, 98.138, 18.233]
  Call Extruder(268.06964)
  MoveL 7580 to (233.75, 162.2, 106.87) mm, rotated rx -180 ry 0 rz -180 deg; joints [-65.549, 63.165, -83.07, 66.852, 98.101, 18.244]
  MoveL 7581 to (233.75, 162.2, 106.87) mm, rotated rx -180 ry 0 rz -180 deg; joints [-65.549, 63.165, -83.07, 66.852, 98.101, 18.244]
  Call Extruder(268.27659)
  MoveL 7582 to (233.45, 162.37, 106.87) mm, rotated rx 180 ry 0 rz -180 deg; joints [-65.662, 63.168, -83.069, 66.959, 98.065, 18.255]
  MoveL 7583 to (233.45, 162.37, 106.87) mm, rotated rx 180 ry 0 rz -180 deg; joints [-65.662, 63.168, -83.069, 66.959, 98.065, 18.255]
  Call Extruder(268.48276)
  MoveL 7584 to (233.14, 162.55, 106.87) mm, rotated rx -180 ry 0 rz 180 deg; joints [-65.774, 63.171, -83.068, 67.066, 98.028, 18.266]
  MoveL 7585 to (233.14, 162.55, 106.87) mm, rotated rx -180 ry 0 rz 180 deg; joints [-65.774, 63.171, -83.068, 67.066, 98.028, 18.266]
  Call Extruder(268.66443)
  MoveL 7586 to (232.87, 162.69, 106.87) mm, rotated rx 180 ry 0 rz 180 deg; joints [-65.874, 63.172, -83.067, 67.162, 97.996, 18.278]
  MoveL 7587 to (232.87, 162.69, 106.87) mm, rotated rx 180 ry 0 rz 180 deg; joints [-65.874, 63.172, -83.067, 67.162, 97.996, 18.278]
  Call Extruder(268.82240)
  MoveL 7588 to (232.62, 162.8, 106.87) mm, rotated rx -180 ry 0 rz 180 deg; joints [-65.961, 63.172, -83.067, 67.246, 97.969, 18.29]
  MoveL 7589 to (232.62, 162.8, 106.87) mm, rotated rx -180 ry 0 rz 180 deg; joints [-65.961, 63.172, -83.067, 67.246, 97.969, 18.29]
  Call Extruder(268.97977)
  MoveL 7590 to (232.37, 162.9, 106.87) mm, rotated rx 180 ry 0 rz 180 deg; joints [-66.048, 63.171, -83.067, 67.329, 97.941, 18.302]
  MoveL 7591 to (232.37, 162.9, 106.87) mm, rotated rx 180 ry 0 rz 180 deg; joints [-66.048, 63.171, -83.067, 67.329, 97.941, 18.302]
  Call Extruder(269.16252)
  MoveL 7592 to (232.08, 163.03, 106.87) mm, rotated rx 180 ry 0 rz -180 deg; joints [-66.149, 63.171, -83.068, 67.426, 97.91, 18.316]
  MoveL 7593 to (232.08, 163.03, 106.87) mm, rotated rx 180 ry 0 rz -180 deg; joints [-66.149, 63.171, -83.068, 67.426, 97.91, 18.316]
  Call Extruder(269.34450)
  MoveL 7594 to (231.78, 163.15, 106.87) mm, rotated rx -180 ry 0 rz -180 deg; joints [-66.251, 63.17, -83.068, 67.524, 97.878, 18.33]
  MoveL 7595 to (231.78, 163.15, 106.87) mm, rotated rx -180 ry 0 rz -180 deg; joints [-66.251, 63.17, -83.068, 67.524, 97.878, 18.33]
  Call Extruder(269.49184)
  MoveL 7596 to (231.54, 163.24, 106.87) mm, rotated rx 180 ry 0 rz -180 deg; joints [-66.333, 63.169, -83.069, 67.603, 97.853, 18.343]
  MoveL 7597 to (231.54, 163.24, 106.87) mm, rotated rx 180 ry 0 rz -180 deg; joints [-66.333, 63.169, -83.069, 67.603, 97.853, 18.343]
  Call Extruder(269.60506)
  MoveL 7598 to (231.35, 163.3, 106.87) mm, rotated rx 180 ry 0 rz -180 deg; joints [-66.397, 63.167, -83.069, 67.664, 97.834, 18.353]
  MoveL 7599 to (231.35, 163.3, 106.87) mm, rotated rx 180 ry 0 rz -180 deg; joints [-66.397, 63.167, -83.069, 67.664, 97.834, 18.353]
  Call Extruder(269.71784)
  MoveL 7600 to (231.17, 163.36, 106.87) mm, rotated rx 180 ry 0 rz 180 deg; joints [-66.46, 63.166, -83.07, 67.725, 97.815, 18.364]
  MoveL 7601 to (231.17, 163.36, 106.87) mm, rotated rx 180 ry 0 rz 180 deg; joints [-66.46, 63.166, -83.07, 67.725, 97.815, 18.364]
  Call Extruder(269.83017)
  MoveL 7602 to (230.98, 163.42, 106.87) mm, rotated rx -180 ry 0 rz 180 deg; joints [-66.524, 63.164, -83.071, 67.786, 97.796, 18.374]
  MoveL 7603 to (230.98, 163.42, 106.87) mm, rotated rx -180 ry 0 rz 180 deg; joints [-66.524, 63.164, -83.071, 67.786, 97.796, 18.374]
  Call Extruder(269.94206)
  MoveL 7604 to (230.79, 163.48, 106.87) mm, rotated rx 180 ry 0 rz -180 deg; joints [-66.587, 63.162, -83.072, 67.847, 97.777, 18.385]
  MoveL 7605 to (230.79, 163.48, 106.87) mm, rotated rx 180 ry 0 rz -180 deg; joints [-66.587, 63.162, -83.072, 67.847, 97.777, 18.385]
  Call Extruder(270.06346)
  MoveL 7606 to (230.58, 163.55, 106.87) mm, rotated rx 180 ry 0 rz 180 deg; joints [-66.656, 63.161, -83.072, 67.914, 97.756, 18.396]
  MoveL 7607 to (230.58, 163.55, 106.87) mm, rotated rx 180 ry 0 rz 180 deg; joints [-66.656, 63.161, -83.072, 67.914, 97.756, 18.396]
  Call Extruder(270.19428)
  MoveL 7608 to (230.36, 163.61, 106.87) mm, rotated rx 180 ry 0 rz 180 deg; joints [-66.731, 63.158, -83.073, 67.986, 97.733, 18.409]
  MoveL 7609 to (230.36, 163.61, 106.87) mm, rotated rx 180 ry 0 rz 180 deg; joints [-66.731, 63.158, -83.073, 67.986, 97.733, 18.409]
  Call Extruder(270.32452)
  MoveL 7610 to (230.14, 163.68, 106.87) mm, rotated rx 180 ry 0 rz 180 deg; joints [-66.805, 63.156, -83.074, 68.058, 97.711, 18.421]
  MoveL 7611 to (230.14, 163.68, 106.87) mm, rotated rx 180 ry 0 rz 180 deg; joints [-66.805, 63.156, -83.074, 68.058, 97.711, 18.421]
  Call Extruder(270.45421)
  MoveL 7612 to (229.91, 163.75, 106.87) mm, rotated rx -180 ry 0 rz -180 deg; joints [-66.88, 63.154, -83.075, 68.13, 97.689, 18.434]
  MoveL 7613 to (229.91, 163.75, 106.87) mm, rotated rx -180 ry 0 rz -180 deg; joints [-66.88, 63.154, -83.075, 68.13, 97.689, 18.434]
  Call Extruder(270.58333)
  MoveL 7614 to (229.69, 163.82, 106.87) mm, rotated rx 180 ry 0 rz -180 deg; joints [-66.955, 63.152, -83.077, 68.202, 97.666, 18.447]
  MoveL 7615 to (229.69, 163.82, 106.87) mm, rotated rx 180 ry 0 rz -180 deg; joints [-66.955, 63.152, -83.077, 68.202, 97.666, 18.447]
  Call Extruder(270.69840)
  MoveL 7616 to (229.48, 163.86, 106.87) mm, rotated rx -180 ry 0 rz 180 deg; joints [-67.021, 63.148, -83.078, 68.266, 97.647, 18.459]
  MoveL 7617 to (229.48, 163.86, 106.87) mm, rotated rx -180 ry 0 rz 180 deg; joints [-67.021, 63.148, -83.078, 68.266, 97.647, 18.459]
  Call Extruder(270.81302)
  MoveL 7618 to (229.28, 163.91, 106.87) mm, rotated rx -180 ry 0 rz 180 deg; joints [-67.087, 63.145, -83.08, 68.329, 97.628, 18.472]
  MoveL 7619 to (229.28, 163.91, 106.87) mm, rotated rx -180 ry 0 rz 180 deg; joints [-67.087, 63.145, -83.08, 68.329, 97.628, 18.472]
  Call Extruder(270.92719)
  MoveL 7620 to (229.08, 163.95, 106.87) mm, rotated rx 180 ry 0 rz -180 deg; joints [-67.153, 63.142, -83.081, 68.393, 97.609, 18.485]
  MoveL 7621 to (229.08, 163.95, 106.87) mm, rotated rx 180 ry 0 rz -180 deg; joints [-67.153, 63.142, -83.081, 68.393, 97.609, 18.485]
  Call Extruder(271.04091)
  MoveL 7622 to (228.87, 164, 106.87) mm, rotated rx -180 ry 0 rz 180 deg; joints [-67.22, 63.139, -83.083, 68.457, 97.589, 18.498]
  MoveL 7623 to (228.87, 164, 106.87) mm, rotated rx -180 ry 0 rz 180 deg; joints [-67.22, 63.139, -83.083, 68.457, 97.589, 18.498]
  Call Extruder(271.16633)
  MoveL 7624 to (228.65, 164.04, 106.87) mm, rotated rx -180 ry 0 rz 180 deg; joints [-67.293, 63.135, -83.084, 68.528, 97.568, 18.512]
  MoveL 7625 to (228.65, 164.04, 106.87) mm, rotated rx -180 ry 0 rz 180 deg; joints [-67.293, 63.135, -83.084, 68.528, 97.568, 18.512]
  Call Extruder(271.30331)
  MoveL 7626 to (228.4, 164.09, 106.87) mm, rotated rx -180 ry 0 rz -180 deg; joints [-67.373, 63.131, -83.086, 68.605, 97.545, 18.528]
  MoveL 7627 to (228.4, 164.09, 106.87) mm, rotated rx -180 ry 0 rz -180 deg; joints [-67.373, 63.131, -83.086, 68.605, 97.545, 18.528]
  Call Extruder(271.43968)
  MoveL 7628 to (228.15, 164.14, 106.87) mm, rotated rx 180 ry 0 rz 180 deg; joints [-67.453, 63.126, -83.088, 68.683, 97.522, 18.544]
  MoveL 7629 to (228.15, 164.14, 106.87) mm, rotated rx 180 ry 0 rz 180 deg; joints [-67.453, 63.126, -83.088, 68.683, 97.522, 18.544]
  Call Extruder(271.57543)
  MoveL 7630 to (227.9, 164.19, 106.87) mm, rotated rx 180 ry 0 rz 180 deg; joints [-67.534, 63.122, -83.09, 68.761, 97.498, 18.56]
  MoveL 7631 to (227.9, 164.19, 106.87) mm, rotated rx 180 ry 0 rz 180 deg; joints [-67.534, 63.122, -83.09, 68.761, 97.498, 18.56]
  Call Extruder(271.71058)
  MoveL 7632 to (227.65, 164.24, 106.87) mm, rotated rx -180 ry 0 rz 180 deg; joints [-67.614, 63.118, -83.092, 68.838, 97.475, 18.576]
  MoveL 7633 to (227.65, 164.24, 106.87) mm, rotated rx -180 ry 0 rz 180 deg; joints [-67.614, 63.118, -83.092, 68.838, 97.475, 18.576]
  Call Extruder(271.84512)
  MoveL 7634 to (227.4, 164.29, 106.87) mm, rotated rx 180 ry 0 rz 180 deg; joints [-67.695, 63.114, -83.094, 68.916, 97.451, 18.591]
  MoveL 7635 to (227.4, 164.29, 106.87) mm, rotated rx 180 ry 0 rz 180 deg; joints [-67.695, 63.114, -83.094, 68.916, 97.451, 18.591]
  Call Extruder(271.97904)
  MoveL 7636 to (227.15, 164.34, 106.87) mm, rotated rx 180 ry 0 rz -180 deg; joints [-67.775, 63.11, -83.096, 68.993, 97.428, 18.607]
  MoveL 7637 to (227.15, 164.34, 106.87) mm, rotated rx 180 ry 0 rz -180 deg; joints [-67.775, 63.11, -83.096, 68.993, 97.428, 18.607]
  Call Extruder(272.12691)
  MoveL 7638 to (226.87, 164.39, 106.87) mm, rotated rx -180 ry 0 rz 180 deg; joints [-67.864, 63.105, -83.098, 69.079, 97.402, 18.625]
  MoveL 7639 to (226.87, 164.39, 106.87) mm, rotated rx -180 ry 0 rz 180 deg; joints [-67.864, 63.105, -83.098, 69.079, 97.402, 18.625]
  Call Extruder(272.28865)
  MoveL 7640 to (226.57, 164.44, 106.87) mm, rotated rx -180 ry 0 rz -180 deg; joints [-67.961, 63.099, -83.101, 69.173, 97.374, 18.645]
  MoveL 7641 to (226.57, 164.44, 106.87) mm, rotated rx -180 ry 0 rz -180 deg; joints [-67.961, 63.099, -83.101, 69.173, 97.374, 18.645]
  Call Extruder(272.44966)
  MoveL 7642 to (226.26, 164.49, 106.87) mm, rotated rx 180 ry 0 rz 180 deg; joints [-68.059, 63.093, -83.104, 69.267, 97.346, 18.665]
  MoveL 7643 to (226.26, 164.49, 106.87) mm, rotated rx 180 ry 0 rz 180 deg; joints [-68.059, 63.093, -83.104, 69.267, 97.346, 18.665]
  Call Extruder(272.60995)
  MoveL 7644 to (225.95, 164.53, 106.87) mm, rotated rx -180 ry 0 rz 180 deg; joints [-68.156, 63.087, -83.106, 69.362, 97.318, 18.685]
  MoveL 7645 to (225.95, 164.53, 106.87) mm, rotated rx -180 ry 0 rz 180 deg; joints [-68.156, 63.087, -83.106, 69.362, 97.318, 18.685]
  Call Extruder(272.76951)
  MoveL 7646 to (225.65, 164.58, 106.87) mm, rotated rx -180 ry 0 rz 180 deg; joints [-68.254, 63.081, -83.109, 69.456, 97.29, 18.705]
  MoveL 7647 to (225.65, 164.58, 106.87) mm, rotated rx -180 ry 0 rz 180 deg; joints [-68.254, 63.081, -83.109, 69.456, 97.29, 18.705]
  Call Extruder(272.92834)
  MoveL 7648 to (225.34, 164.63, 106.87) mm, rotated rx 180 ry 0 rz -180 deg; joints [-68.351, 63.076, -83.112, 69.55, 97.261, 18.724]
  MoveL 7649 to (225.34, 164.63, 106.87) mm, rotated rx 180 ry 0 rz -180 deg; joints [-68.351, 63.076, -83.112, 69.55, 97.261, 18.724]
  Call Extruder(273.10701)
  MoveL 7650 to (225, 164.68, 106.87) mm, rotated rx -180 ry 0 rz 180 deg; joints [-68.461, 63.068, -83.115, 69.656, 97.23, 18.748]
  MoveL 7651 to (225, 164.68, 106.87) mm, rotated rx -180 ry 0 rz 180 deg; joints [-68.461, 63.068, -83.115, 69.656, 97.23, 18.748]
  Call Extruder(273.30545)
  MoveL 7652 to (224.61, 164.72, 106.87) mm, rotated rx 180 ry 0 rz 180 deg; joints [-68.583, 63.06, -83.119, 69.774, 97.195, 18.774]
  MoveL 7653 to (224.61, 164.72, 106.87) mm, rotated rx 180 ry 0 rz 180 deg; joints [-68.583, 63.06, -83.119, 69.774, 97.195, 18.774]
  Call Extruder(273.50302)
  MoveL 7654 to (224.22, 164.77, 106.87) mm, rotated rx -180 ry 0 rz -180 deg; joints [-68.706, 63.052, -83.122, 69.893, 97.159, 18.8]
  MoveL 7655 to (224.22, 164.77, 106.87) mm, rotated rx -180 ry 0 rz -180 deg; joints [-68.706, 63.052, -83.122, 69.893, 97.159, 18.8]
  Call Extruder(273.69973)
  MoveL 7656 to (223.84, 164.82, 106.87) mm, rotated rx -180 ry 0 rz 180 deg; joints [-68.828, 63.043, -83.126, 70.011, 97.124, 18.826]
  MoveL 7657 to (223.84, 164.82, 106.87) mm, rotated rx -180 ry 0 rz 180 deg; joints [-68.828, 63.043, -83.126, 70.011, 97.124, 18.826]
  Call Extruder(273.89557)
  MoveL 7658 to (223.45, 164.86, 106.87) mm, rotated rx 180 ry 0 rz -180 deg; joints [-68.951, 63.035, -83.13, 70.129, 97.088, 18.852]
  MoveL 7659 to (223.45, 164.86, 106.87) mm, rotated rx 180 ry 0 rz -180 deg; joints [-68.951, 63.035, -83.13, 70.129, 97.088, 18.852]
  Call Extruder(274.19092)
  MoveL 7660 to (222.86, 164.91, 106.87) mm, rotated rx -180 ry 0 rz -180 deg; joints [-69.135, 63.021, -83.136, 70.307, 97.036, 18.893]
  MoveL 7661 to (222.86, 164.91, 106.87) mm, rotated rx -180 ry 0 rz -180 deg; joints [-69.135, 63.021, -83.136, 70.307, 97.036, 18.893]
  Call Extruder(274.48494)
  MoveL 7662 to (222.27, 164.95, 106.87) mm, rotated rx -180 ry 0 rz 180 deg; joints [-69.319, 63.007, -83.143, 70.485, 96.983, 18.934]
  MoveL 7663 to (222.27, 164.95, 106.87) mm, rotated rx -180 ry 0 rz 180 deg; joints [-69.319, 63.007, -83.143, 70.485, 96.983, 18.934]
  Call Extruder(274.77764)
  MoveL 7664 to (221.68, 165, 106.87) mm, rotated rx 180 ry 0 rz 180 deg; joints [-69.504, 62.993, -83.149, 70.663, 96.93, 18.974]
  MoveL 7665 to (221.68, 165, 106.87) mm, rotated rx 180 ry 0 rz 180 deg; joints [-69.504, 62.993, -83.149, 70.663, 96.93, 18.974]
  Call Extruder(275.35108)
  MoveL 7666 to (220.52, 165.05, 106.87) mm, rotated rx -180 ry 0 rz 180 deg; joints [-69.864, 62.962, -83.163, 71.011, 96.827, 19.058]
  MoveL 7667 to (220.52, 165.05, 106.87) mm, rotated rx -180 ry 0 rz 180 deg; joints [-69.864, 62.962, -83.163, 71.011, 96.827, 19.058]
  Call Extruder(276.06510)
  MoveL 7668 to (219.06, 165.09, 106.87) mm, rotated rx -180 ry 0 rz 180 deg; joints [-70.315, 62.923, -83.18, 71.447, 96.698, 19.162]
  Call Extruder(392.91185)
  MoveL 7669 to (-19.06, 165.09, 106.87) mm, rotated rx -180 ry 0 rz 180 deg; joints [-137.325, 68.044, -79.702, 136.73, 81.457, 7.961]
  Call Extruder(393.34045)
  MoveL 7670 to (-19.94, 165.07, 106.87) mm, rotated rx 180 ry 0 rz 180 deg; joints [-137.467, 68.085, -79.661, 136.88, 81.496, 7.884]
  MoveL 7671 to (-19.94, 165.07, 106.87) mm, rotated rx 180 ry 0 rz 180 deg; joints [-137.467, 68.085, -79.661, 136.88, 81.496, 7.884]
  Call Extruder(393.91390)
  MoveL 7672 to (-21.1, 165.03, 106.87) mm, rotated rx 180 ry 0 rz -180 deg; joints [-137.659, 68.138, -79.608, 137.083, 81.548, 7.782]
  MoveL 7673 to (-21.1, 165.03, 106.87) mm, rotated rx 180 ry 0 rz -180 deg; joints [-137.659, 68.138, -79.608, 137.083, 81.548, 7.782]
  Call Extruder(394.34820)
  MoveL 7674 to (-21.97, 164.98, 106.87) mm, rotated rx 180 ry 0 rz 180 deg; joints [-137.804, 68.177, -79.568, 137.237, 81.586, 7.707]
  MoveL 7675 to (-21.97, 164.98, 106.87) mm, rotated rx 180 ry 0 rz 180 deg; joints [-137.804, 68.177, -79.568, 137.237, 81.586, 7.707]
  Call Extruder(394.64223)
  MoveL 7676 to (-22.56, 164.93, 106.87) mm, rotated rx 180 ry 0 rz -180 deg; joints [-137.905, 68.203, -79.542, 137.342, 81.611, 7.656]
  MoveL 7677 to (-22.56, 164.93, 106.87) mm, rotated rx 180 ry 0 rz -180 deg; joints [-137.905, 68.203, -79.542, 137.342, 81.611, 7.656]
  Call Extruder(394.93759)
  MoveL 7678 to (-23.15, 164.89, 106.87) mm, rotated rx -180 ry 0 rz 180 deg; joints [-138.004, 68.229, -79.516, 137.447, 81.636, 7.606]
  MoveL 7679 to (-23.15, 164.89, 106.87) mm, rotated rx -180 ry 0 rz 180 deg; joints [-138.004, 68.229, -79.516, 137.447, 81.636, 7.606]
  Call Extruder(395.18380)
  MoveL 7680 to (-23.64, 164.84, 106.87) mm, rotated rx -180 ry 0 rz 180 deg; joints [-138.088, 68.25, -79.494, 137.536, 81.657, 7.565]
  MoveL 7681 to (-23.64, 164.84, 106.87) mm, rotated rx -180 ry 0 rz 180 deg; joints [-138.088, 68.25, -79.494, 137.536, 81.657, 7.565]
  Call Extruder(395.38051)
  MoveL 7682 to (-24.03, 164.79, 106.87) mm, rotated rx 180 ry 0 rz -180 deg; joints [-138.156, 68.266, -79.477, 137.607, 81.672, 7.532]
  MoveL 7683 to (-24.03, 164.79, 106.87) mm, rotated rx 180 ry 0 rz -180 deg; joints [-138.156, 68.266, -79.477, 137.607, 81.672, 7.532]
  Call Extruder(395.57808)
  MoveL 7684 to (-24.42, 164.75, 106.87) mm, rotated rx 180 ry 0 rz 180 deg; joints [-138.224, 68.283, -79.46, 137.678, 81.688, 7.5]
  MoveL 7685 to (-24.42, 164.75, 106.87) mm, rotated rx 180 ry 0 rz 180 deg; joints [-138.224, 68.283, -79.46, 137.678, 81.688, 7.5]
  Call Extruder(395.77652)
  MoveL 7686 to (-24.8, 164.7, 106.87) mm, rotated rx -180 ry 0 rz 180 deg; joints [-138.292, 68.299, -79.444, 137.749, 81.703, 7.467]
  MoveL 7687 to (-24.8, 164.7, 106.87) mm, rotated rx -180 ry 0 rz 180 deg; joints [-138.292, 68.299, -79.444, 137.749, 81.703, 7.467]
  Call Extruder(395.97583)
  MoveL 7688 to (-25.19, 164.66, 106.87) mm, rotated rx 180 ry 0 rz 180 deg; joints [-138.359, 68.315, -79.427, 137.82, 81.719, 7.435]
  MoveL 7689 to (-25.19, 164.66, 106.87) mm, rotated rx 180 ry 0 rz 180 deg; joints [-138.359, 68.315, -79.427, 137.82, 81.719, 7.435]
  Call Extruder(396.13466)
  MoveL 7690 to (-25.5, 164.61, 106.87) mm, rotated rx -180 ry 0 rz -180 deg; joints [-138.415, 68.328, -79.414, 137.878, 81.731, 7.41]
  MoveL 7691 to (-25.5, 164.61, 106.87) mm, rotated rx -180 ry 0 rz -180 deg; joints [-138.415, 68.328, -79.414, 137.878, 81.731, 7.41]
  Call Extruder(396.29423)
  MoveL 7692 to (-25.8, 164.56, 106.87) mm, rotated rx -180 ry 0 rz 180 deg; joints [-138.47, 68.34, -79.401, 137.936, 81.742, 7.385]
  MoveL 7693 to (-25.8, 164.56, 106.87) mm, rotated rx -180 ry 0 rz 180 deg; joints [-138.47, 68.34, -79.401, 137.936, 81.742, 7.385]
  Call Extruder(396.45451)
  MoveL 7694 to (-26.11, 164.51, 106.87) mm, rotated rx 180 ry 0 rz 180 deg; joints [-138.525, 68.352, -79.388, 137.994, 81.754, 7.36]
  MoveL 7695 to (-26.11, 164.51, 106.87) mm, rotated rx 180 ry 0 rz 180 deg; joints [-138.525, 68.352, -79.388, 137.994, 81.754, 7.36]
  Call Extruder(396.61553)
  MoveL 7696 to (-26.41, 164.46, 106.87) mm, rotated rx 180 ry 0 rz -180 deg; joints [-138.58, 68.365, -79.375, 138.051, 81.766, 7.335]
  MoveL 7697 to (-26.41, 164.46, 106.87) mm, rotated rx 180 ry 0 rz -180 deg; joints [-138.58, 68.365, -79.375, 138.051, 81.766, 7.335]
  Call Extruder(396.77727)
  MoveL 7698 to (-26.72, 164.41, 106.87) mm, rotated rx -180 ry 0 rz -180 deg; joints [-138.635, 68.377, -79.362, 138.109, 81.778, 7.31]
  MoveL 7699 to (-26.72, 164.41, 106.87) mm, rotated rx -180 ry 0 rz -180 deg; joints [-138.635, 68.377, -79.362, 138.109, 81.778, 7.31]
  Call Extruder(396.93974)
  MoveL 7700 to (-27.03, 164.37, 106.87) mm, rotated rx 180 ry 0 rz -180 deg; joints [-138.69, 68.389, -79.349, 138.166, 81.79, 7.285]
  MoveL 7701 to (-27.03, 164.37, 106.87) mm, rotated rx 180 ry 0 rz -180 deg; joints [-138.69, 68.389, -79.349, 138.166, 81.79, 7.285]
  Call Extruder(397.07367)
  MoveL 7702 to (-27.28, 164.32, 106.87) mm, rotated rx 180 ry 0 rz 180 deg; joints [-138.736, 68.399, -79.339, 138.215, 81.799, 7.265]
  MoveL 7703 to (-27.28, 164.32, 106.87) mm, rotated rx 180 ry 0 rz 180 deg; joints [-138.736, 68.399, -79.339, 138.215, 81.799, 7.265]
  Call Extruder(397.20821)
  MoveL 7704 to (-27.52, 164.27, 106.87) mm, rotated rx 180 ry 0 rz 180 deg; joints [-138.783, 68.409, -79.329, 138.263, 81.808, 7.245]
  MoveL 7705 to (-27.52, 164.27, 106.87) mm, rotated rx 180 ry 0 rz 180 deg; joints [-138.783, 68.409, -79.329, 138.263, 81.808, 7.245]
  Call Extruder(397.34335)
  MoveL 7706 to (-27.77, 164.22, 106.87) mm, rotated rx -180 ry 0 rz 180 deg; joints [-138.829, 68.418, -79.318, 138.311, 81.817, 7.225]
  MoveL 7707 to (-27.77, 164.22, 106.87) mm, rotated rx -180 ry 0 rz 180 deg; joints [-138.829, 68.418, -79.318, 138.311, 81.817, 7.225]
  Call Extruder(397.47911)
  MoveL 7708 to (-28.02, 164.17, 106.87) mm, rotated rx -180 ry 0 rz 180 deg; joints [-138.875, 68.428, -79.308, 138.359, 81.826, 7.205]
  MoveL 7709 to (-28.02, 164.17, 106.87) mm, rotated rx -180 ry 0 rz 180 deg; joints [-138.875, 68.428, -79.308, 138.359, 81.826, 7.205]
  Call Extruder(397.61548)
  MoveL 7710 to (-28.27, 164.12, 106.87) mm, rotated rx -180 ry 0 rz 180 deg; joints [-138.921, 68.438, -79.298, 138.408, 81.835, 7.185]
  MoveL 7711 to (-28.27, 164.12, 106.87) mm, rotated rx -180 ry 0 rz 180 deg; joints [-138.921, 68.438, -79.298, 138.408, 81.835, 7.185]
  Call Extruder(397.70034)
  MoveL 7712 to (-28.42, 164.09, 106.87) mm, rotated rx -180 ry 0 rz 180 deg; joints [-138.95, 68.444, -79.292, 138.437, 81.84, 7.173]
  Set speed (130.0 mm/s)
  MoveL 7713 to (-31.76, 163.31, 106.87) mm, rotated rx 180 ry 0 rz -180 deg; joints [-139.581, 68.569, -79.157, 139.095, 81.958, 6.911]
  MoveL 7714 to (-31.76, 163.31, 116.27) mm, rotated rx 180 ry 0 rz 180 deg; joints [-139.581, 69.926, -80.975, 139.051, 81.61, 7.216]
  Call Extruder(395.70034)
  Set speed (40.0 mm/s)
  MoveL 7715 to (-31.76, 163.31, 116.27) mm, rotated rx 180 ry 0 rz 180 deg; joints [-139.581, 69.926, -80.975, 139.051, 81.61, 7.216]
  Call Extruder(0.00000)
  Set speed (130.0 mm/s)
  MoveL 7716 to (-34.23, 161.92, 116.27) mm, rotated rx -180 ry 0 rz -180 deg; joints [-140.182, 69.988, -80.908, 139.667, 81.633, 7.043]
  Call Extruder(2.00000)
  Set speed (40.0 mm/s)
  MoveL 7717 to (-34.23, 161.92, 116.27) mm, rotated rx -180 ry 0 rz -180 deg; joints [-140.182, 69.988, -80.908, 139.667, 81.633, 7.043]
  Set speed (30.0 mm/s)
  MoveL 7718 to (-34.23, 161.92, 116.27) mm, rotated rx -180 ry 0 rz -180 deg; joints [-140.182, 69.988, -80.908, 139.667, 81.633, 7.043]
  Call Extruder(2.16612)
  MoveL 7719 to (-34.45, 161.76, 116.27) mm, rotated rx -180 ry 0 rz -180 deg; joints [-140.244, 69.992, -80.903, 139.729, 81.633, 7.028]
  MoveL 7720 to (-34.45, 161.76, 116.27) mm, rotated rx -180 ry 0 rz -180 deg; joints [-140.244, 69.992, -80.903, 139.729, 81.633, 7.028]
  Call Extruder(2.49954)
  MoveL 7721 to (-34.9, 161.43, 116.27) mm, rotated rx -180 ry 0 rz 180 deg; joints [-140.366, 70.001, -80.894, 139.854, 81.631, 6.999]
  MoveL 7722 to (-34.9, 161.43, 116.27) mm, rotated rx -180 ry 0 rz 180 deg; joints [-140.366, 70.001, -80.894, 139.854, 81.631, 6.999]
  Call Extruder(2.83415)
  MoveL 7723 to (-35.35, 161.1, 116.27) mm, rotated rx -180 ry 0 rz -180 deg; joints [-140.489, 70.01, -80.885, 139.978, 81.63, 6.969]
  Call Extruder(3.66207)
  MoveL 7724 to (-36.39, 160.19, 116.27) mm, rotated rx 180 ry 0 rz 180 deg; joints [-140.797, 70.024, -80.87, 140.29, 81.615, 6.905]
  Call Extruder(4.49000)
  MoveL 7725 to (-37.3, 159.15, 116.27) mm, rotated rx 180 ry 0 rz 180 deg; joints [-141.109, 70.027, -80.866, 140.604, 81.584, 6.855]
  Call Extruder(4.65731)
  MoveL 7726 to (-37.47, 158.93, 116.27) mm, rotated rx 180 ry 0 rz 180 deg; joints [-141.172, 70.026, -80.867, 140.667, 81.575, 6.847]
  MoveL 7727 to (-37.47, 158.93, 116.27) mm, rotated rx 180 ry 0 rz 180 deg; joints [-141.172, 70.026, -80.867, 140.667, 81.575, 6.847]
  Call Extruder(4.99074)
  MoveL 7728 to (-37.8, 158.48, 116.27) mm, rotated rx 180 ry 0 rz 180 deg; joints [-141.298, 70.024, -80.869, 140.793, 81.557, 6.83]
  MoveL 7729 to (-37.8, 158.48, 116.27) mm, rotated rx 180 ry 0 rz 180 deg; joints [-141.298, 70.024, -80.869, 140.793, 81.557, 6.83]
  Call Extruder(5.32299)
  MoveL 7730 to (-38.12, 158.02, 116.27) mm, rotated rx -180 ry 0 rz 180 deg; joints [-141.424, 70.023, -80.87, 140.919, 81.539, 6.814]
  MoveL 7731 to (-38.12, 158.02, 116.27) mm, rotated rx -180 ry 0 rz 180 deg; joints [-141.424, 70.023, -80.87, 140.919, 81.539, 6.814]
  Call Extruder(5.44066)
  MoveL 7732 to (-38.22, 157.85, 116.27) mm, rotated rx 180 ry 0 rz 180 deg; joints [-141.468, 70.021, -80.872, 140.963, 81.531, 6.81]
  MoveL 7733 to (-38.22, 157.85, 116.27) mm, rotated rx 180 ry 0 rz 180 deg; joints [-141.468, 70.021, -80.872, 140.963, 81.531, 6.81]
  Call Extruder(5.64838)
  MoveL 7734 to (-38.4, 157.55, 116.27) mm, rotated rx -180 ry 0 rz 180 deg; joints [-141.547, 70.018, -80.876, 141.042, 81.517, 6.802]
  MoveL 7735 to (-38.4, 157.55, 116.27) mm, rotated rx -180 ry 0 rz 180 deg; joints [-141.547, 70.018, -80.876, 141.042, 81.517, 6.802]
  Call Extruder(5.85533)
  MoveL 7736 to (-38.57, 157.25, 116.27) mm, rotated rx -180 ry 0 rz 180 deg; joints [-141.625, 70.015, -80.879, 141.12, 81.502, 6.795]
  MoveL 7737 to (-38.57, 157.25, 116.27) mm, rotated rx -180 ry 0 rz 180 deg; joints [-141.625, 70.015, -80.879, 141.12, 81.502, 6.795]
  Call Extruder(6.06150)
  MoveL 7738 to (-38.75, 156.94, 116.27) mm, rotated rx 180 ry 0 rz 180 deg; joints [-141.704, 70.011, -80.883, 141.198, 81.488, 6.787]
  MoveL 7739 to (-38.75, 156.94, 116.27) mm, rotated rx 180 ry 0 rz 180 deg; joints [-141.704, 70.011, -80.883, 141.198, 81.488, 6.787]
  Call Extruder(6.24318)
  MoveL 7740 to (-38.89, 156.66, 116.27) mm, rotated rx 180 ry 0 rz -180 deg; joints [-141.773, 70.008, -80.887, 141.267, 81.474, 6.782]
  MoveL 7741 to (-38.89, 156.66, 116.27) mm, rotated rx 180 ry 0 rz -180 deg; joints [-141.773, 70.008, -80.887, 141.267, 81.474, 6.782]
  Call Extruder(6.40116)
  MoveL 7742 to (-39, 156.42, 116.27) mm, rotated rx -180 ry 0 rz 180 deg; joints [-141.832, 70.003, -80.892, 141.325, 81.459, 6.779]
  MoveL 7743 to (-39, 156.42, 116.27) mm, rotated rx -180 ry 0 rz 180 deg; joints [-141.832, 70.003, -80.892, 141.325, 81.459, 6.779]
  Call Extruder(6.55855)
  MoveL 7744 to (-39.11, 156.17, 116.27) mm, rotated rx 180 ry 0 rz -180 deg; joints [-141.891, 69.999, -80.896, 141.384, 81.445, 6.776]
  MoveL 7745 to (-39.11, 156.17, 116.27) mm, rotated rx 180 ry 0 rz -180 deg; joints [-141.891, 69.999, -80.896, 141.384, 81.445, 6.776]
  Call Extruder(6.74127)
  MoveL 7746 to (-39.22, 155.87, 116.27) mm, rotated rx -180 ry 0 rz 180 deg; joints [-141.96, 69.994, -80.902, 141.452, 81.429, 6.773]
  MoveL 7747 to (-39.22, 155.87, 116.27) mm, rotated rx -180 ry 0 rz 180 deg; joints [-141.96, 69.994, -80.902, 141.452, 81.429, 6.773]
  Call Extruder(6.92323)
  MoveL 7748 to (-39.35, 155.58, 116.27) mm, rotated rx -180 ry 0 rz 180 deg; joints [-142.029, 69.988, -80.908, 141.52, 81.412, 6.769]
  MoveL 7749 to (-39.35, 155.58, 116.27) mm, rotated rx -180 ry 0 rz 180 deg; joints [-142.029, 69.988, -80.908, 141.52, 81.412, 6.769]
  Call Extruder(7.07056)
  MoveL 7750 to (-39.44, 155.34, 116.27) mm, rotated rx -180 ry 0 rz 180 deg; joints [-142.085, 69.984, -80.913, 141.575, 81.398, 6.767]
  MoveL 7751 to (-39.44, 155.34, 116.27) mm, rotated rx -180 ry 0 rz 180 deg; joints [-142.085, 69.984, -80.913, 141.575, 81.398, 6.767]
  Call Extruder(7.18380)
  MoveL 7752 to (-39.5, 155.15, 116.27) mm, rotated rx -180 ry 0 rz 180 deg; joints [-142.127, 69.979, -80.917, 141.617, 81.386, 6.766]
  MoveL 7753 to (-39.5, 155.15, 116.27) mm, rotated rx -180 ry 0 rz 180 deg; joints [-142.127, 69.979, -80.917, 141.617, 81.386, 6.766]
  Call Extruder(7.29659)
  MoveL 7754 to (-39.56, 154.97, 116.27) mm, rotated rx 180 ry 0 rz 180 deg; joints [-142.169, 69.975, -80.922, 141.658, 81.374, 6.765]
  MoveL 7755 to (-39.56, 154.97, 116.27) mm, rotated rx 180 ry 0 rz 180 deg; joints [-142.169, 69.975, -80.922, 141.658, 81.374, 6.765]
  Call Extruder(7.40893)
  MoveL 7756 to (-39.62, 154.78, 116.27) mm, rotated rx 180 ry 0 rz 180 deg; joints [-142.212, 69.971, -80.926, 141.7, 81.362, 6.764]
  MoveL 7757 to (-39.62, 154.78, 116.27) mm, rotated rx 180 ry 0 rz 180 deg; joints [-142.212, 69.971, -80.926, 141.7, 81.362, 6.764]
  Call Extruder(7.52083)
  MoveL 7758 to (-39.68, 154.59, 116.27) mm, rotated rx 180 ry 0 rz 180 deg; joints [-142.254, 69.967, -80.931, 141.742, 81.35, 6.763]
  MoveL 7759 to (-39.68, 154.59, 116.27) mm, rotated rx 180 ry 0 rz 180 deg; joints [-142.254, 69.967, -80.931, 141.742, 81.35, 6.763]
  Call Extruder(7.64223)
  MoveL 7760 to (-39.75, 154.38, 116.27) mm, rotated rx -180 ry 0 rz -180 deg; joints [-142.3, 69.962, -80.936, 141.787, 81.337, 6.763]
  MoveL 7761 to (-39.75, 154.38, 116.27) mm, rotated rx -180 ry 0 rz -180 deg; joints [-142.3, 69.962, -80.936, 141.787, 81.337, 6.763]
  Call Extruder(7.77303)
  MoveL 7762 to (-39.81, 154.16, 116.27) mm, rotated rx -180 ry 0 rz 180 deg; joints [-142.35, 69.957, -80.942, 141.836, 81.323, 6.762]
  MoveL 7763 to (-39.81, 154.16, 116.27) mm, rotated rx -180 ry 0 rz 180 deg; joints [-142.35, 69.957, -80.942, 141.836, 81.323, 6.762]
  Call Extruder(7.90326)
  MoveL 7764 to (-39.88, 153.94, 116.27) mm, rotated rx -180 ry 0 rz 180 deg; joints [-142.399, 69.952, -80.947, 141.885, 81.309, 6.761]
  MoveL 7765 to (-39.88, 153.94, 116.27) mm, rotated rx -180 ry 0 rz 180 deg; joints [-142.399, 69.952, -80.947, 141.885, 81.309, 6.761]
  Call Extruder(8.03292)
  MoveL 7766 to (-39.95, 153.71, 116.27) mm, rotated rx 180 ry 0 rz -180 deg; joints [-142.449, 69.946, -80.953, 141.933, 81.294, 6.76]
  MoveL 7767 to (-39.95, 153.71, 116.27) mm, rotated rx 180 ry 0 rz -180 deg; joints [-142.449, 69.946, -80.953, 141.933, 81.294, 6.76]
  Call Extruder(8.16202)
  MoveL 7768 to (-40.02, 153.49, 116.27) mm, rotated rx 180 ry 0 rz -180 deg; joints [-142.498, 69.941, -80.958, 141.982, 81.28, 6.759]
  MoveL 7769 to (-40.02, 153.49, 116.27) mm, rotated rx 180 ry 0 rz -180 deg; joints [-142.498, 69.941, -80.958, 141.982, 81.28, 6.759]
  Call Extruder(8.27711)
  MoveL 7770 to (-40.06, 153.28, 116.27) mm, rotated rx 180 ry 0 rz 180 deg; joints [-142.541, 69.936, -80.964, 142.024, 81.266, 6.76]
  MoveL 7771 to (-40.06, 153.28, 116.27) mm, rotated rx 180 ry 0 rz 180 deg; joints [-142.541, 69.936, -80.964, 142.024, 81.266, 6.76]
  Call Extruder(8.39175)
  MoveL 7772 to (-40.11, 153.08, 116.27) mm, rotated rx 180 ry 0 rz 180 deg; joints [-142.584, 69.93, -80.97, 142.067, 81.252, 6.761]
  MoveL 7773 to (-40.11, 153.08, 116.27) mm, rotated rx 180 ry 0 rz 180 deg; joints [-142.584, 69.93, -80.97, 142.067, 81.252, 6.761]
  Call Extruder(8.50593)
  MoveL 7774 to (-40.15, 152.88, 116.27) mm, rotated rx 180 ry 0 rz -180 deg; joints [-142.627, 69.924, -80.976, 142.109, 81.237, 6.761]
  MoveL 7775 to (-40.15, 152.88, 116.27) mm, rotated rx 180 ry 0 rz -180 deg; joints [-142.627, 69.924, -80.976, 142.109, 81.237, 6.761]
  Call Extruder(8.61966)
  MoveL 7776 to (-40.2, 152.67, 116.27) mm, rotated rx 180 ry 0 rz 180 deg; joints [-142.671, 69.919, -80.982, 142.151, 81.223, 6.762]
  MoveL 7777 to (-40.2, 152.67, 116.27) mm, rotated rx 180 ry 0 rz 180 deg; joints [-142.671, 69.919, -80.982, 142.151, 81.223, 6.762]
  Call Extruder(8.74509)
  MoveL 7778 to (-40.24, 152.45, 116.27) mm, rotated rx -180 ry 0 rz -180 deg; joints [-142.718, 69.913, -80.989, 142.197, 81.207, 6.762]
  MoveL 7779 to (-40.24, 152.45, 116.27) mm, rotated rx -180 ry 0 rz -180 deg; joints [-142.718, 69.913, -80.989, 142.197, 81.207, 6.762]
  Call Extruder(8.88206)
  MoveL 7780 to (-40.29, 152.2, 116.27) mm, rotated rx 180 ry 0 rz 180 deg; joints [-142.77, 69.906, -80.996, 142.249, 81.19, 6.763]
  MoveL 7781 to (-40.29, 152.2, 116.27) mm, rotated rx 180 ry 0 rz 180 deg; joints [-142.77, 69.906, -80.996, 142.249, 81.19, 6.763]
  Call Extruder(9.01843)
  MoveL 7782 to (-40.34, 151.95, 116.27) mm, rotated rx -180 ry 0 rz -180 deg; joints [-142.822, 69.899, -81.004, 142.299, 81.172, 6.764]
  MoveL 7783 to (-40.34, 151.95, 116.27) mm, rotated rx -180 ry 0 rz -180 deg; joints [-142.822, 69.899, -81.004, 142.299, 81.172, 6.764]
  Call Extruder(9.15418)
  MoveL 7784 to (-40.39, 151.7, 116.27) mm, rotated rx -180 ry 0 rz 180 deg; joints [-142.874, 69.892, -81.011, 142.35, 81.155, 6.765]
  MoveL 7785 to (-40.39, 151.7, 116.27) mm, rotated rx -180 ry 0 rz 180 deg; joints [-142.874, 69.892, -81.011, 142.35, 81.155, 6.765]
  Call Extruder(9.28933)
  MoveL 7786 to (-40.44, 151.45, 116.27) mm, rotated rx -180 ry 0 rz 180 deg; joints [-142.926, 69.885, -81.018, 142.401, 81.137, 6.766]
  MoveL 7787 to (-40.44, 151.45, 116.27) mm, rotated rx -180 ry 0 rz 180 deg; joints [-142.926, 69.885, -81.018, 142.401, 81.137, 6.766]
  Call Extruder(9.42386)
  MoveL 7788 to (-40.49, 151.2, 116.27) mm, rotated rx 180 ry 0 rz 180 deg; joints [-142.978, 69.878, -81.026, 142.452, 81.12, 6.767]
  MoveL 7789 to (-40.49, 151.2, 116.27) mm, rotated rx 180 ry 0 rz 180 deg; joints [-142.978, 69.878, -81.026, 142.452, 81.12, 6.767]
  Call Extruder(9.55779)
  MoveL 7790 to (-40.54, 150.95, 116.27) mm, rotated rx -180 ry 0 rz 180 deg; joints [-143.031, 69.871, -81.033, 142.503, 81.102, 6.768]
  MoveL 7791 to (-40.54, 150.95, 116.27) mm, rotated rx -180 ry 0 rz 180 deg; joints [-143.031, 69.871, -81.033, 142.503, 81.102, 6.768]
  Call Extruder(9.70564)
  MoveL 7792 to (-40.59, 150.67, 116.27) mm, rotated rx 180 ry 0 rz 180 deg; joints [-143.088, 69.863, -81.042, 142.559, 81.082, 6.769]
  MoveL 7793 to (-40.59, 150.67, 116.27) mm, rotated rx 180 ry 0 rz 180 deg; joints [-143.088, 69.863, -81.042, 142.559, 81.082, 6.769]
  Call Extruder(9.86737)
  MoveL 7794 to (-40.64, 150.37, 116.27) mm, rotated rx 180 ry 0 rz 180 deg; joints [-143.15, 69.853, -81.051, 142.621, 81.06, 6.771]
  MoveL 7795 to (-40.64, 150.37, 116.27) mm, rotated rx 180 ry 0 rz 180 deg; joints [-143.15, 69.853, -81.051, 142.621, 81.06, 6.771]
  Call Extruder(10.02836)
  MoveL 7796 to (-40.69, 150.06, 116.27) mm, rotated rx -180 ry 0 rz 180 deg; joints [-143.213, 69.844, -81.061, 142.682, 81.038, 6.772]
  MoveL 7797 to (-40.69, 150.06, 116.27) mm, rotated rx -180 ry 0 rz 180 deg; joints [-143.213, 69.844, -81.061, 142.682, 81.038, 6.772]
  Call Extruder(10.18863)
  MoveL 7798 to (-40.74, 149.76, 116.27) mm, rotated rx -180 ry 0 rz 180 deg; joints [-143.276, 69.835, -81.071, 142.743, 81.015, 6.774]
  MoveL 7799 to (-40.74, 149.76, 116.27) mm, rotated rx -180 ry 0 rz 180 deg; joints [-143.276, 69.835, -81.071, 142.743, 81.015, 6.774]
  Call Extruder(10.34817)
  MoveL 7800 to (-40.78, 149.45, 116.27) mm, rotated rx 180 ry 0 rz 180 deg; joints [-143.338, 69.826, -81.08, 142.804, 80.993, 6.776]
  MoveL 7801 to (-40.78, 149.45, 116.27) mm, rotated rx 180 ry 0 rz 180 deg; joints [-143.338, 69.826, -81.08, 142.804, 80.993, 6.776]
  Call Extruder(10.50698)
  MoveL 7802 to (-40.83, 149.14, 116.27) mm, rotated rx -180 ry 0 rz -180 deg; joints [-143.401, 69.817, -81.09, 142.866, 80.971, 6.777]
  MoveL 7803 to (-40.83, 149.14, 116.27) mm, rotated rx -180 ry 0 rz -180 deg; joints [-143.401, 69.817, -81.09, 142.866, 80.971, 6.777]
  Call Extruder(10.68565)
  MoveL 7804 to (-40.88, 148.8, 116.27) mm, rotated rx 180 ry 0 rz -180 deg; joints [-143.471, 69.806, -81.101, 142.934, 80.945, 6.779]
  MoveL 7805 to (-40.88, 148.8, 116.27) mm, rotated rx 180 ry 0 rz -180 deg; joints [-143.471, 69.806, -81.101, 142.934, 80.945, 6.779]
  Call Extruder(10.88409)
  MoveL 7806 to (-40.93, 148.41, 116.27) mm, rotated rx -180 ry 0 rz 180 deg; joints [-143.549, 69.794, -81.114, 143.01, 80.916, 6.782]
  MoveL 7807 to (-40.93, 148.41, 116.27) mm, rotated rx -180 ry 0 rz 180 deg; joints [-143.549, 69.794, -81.114, 143.01, 80.916, 6.782]
  Call Extruder(11.08166)
  MoveL 7808 to (-40.97, 148.02, 116.27) mm, rotated rx -180 ry 0 rz -180 deg; joints [-143.627, 69.782, -81.126, 143.086, 80.887, 6.785]
  MoveL 7809 to (-40.97, 148.02, 116.27) mm, rotated rx -180 ry 0 rz -180 deg; joints [-143.627, 69.782, -81.126, 143.086, 80.887, 6.785]
  Call Extruder(11.27837)
  MoveL 7810 to (-41.02, 147.63, 116.27) mm, rotated rx -180 ry 0 rz 180 deg; joints [-143.705, 69.769, -81.139, 143.162, 80.857, 6.788]
  MoveL 7811 to (-41.02, 147.63, 116.27) mm, rotated rx -180 ry 0 rz 180 deg; joints [-143.705, 69.769, -81.139, 143.162, 80.857, 6.788]
  Call Extruder(11.47421)
  MoveL 7812 to (-41.06, 147.25, 116.27) mm, rotated rx 180 ry 0 rz 180 deg; joints [-143.783, 69.757, -81.152, 143.237, 80.828, 6.791]
  MoveL 7813 to (-41.06, 147.25, 116.27) mm, rotated rx 180 ry 0 rz 180 deg; joints [-143.783, 69.757, -81.152, 143.237, 80.828, 6.791]
  Call Extruder(11.76961)
  MoveL 7814 to (-41.11, 146.66, 116.27) mm, rotated rx -180 ry 0 rz -180 deg; joints [-143.899, 69.737, -81.172, 143.35, 80.782, 6.797]
  MoveL 7815 to (-41.11, 146.66, 116.27) mm, rotated rx -180 ry 0 rz -180 deg; joints [-143.899, 69.737, -81.172, 143.35, 80.782, 6.797]
  Call Extruder(12.06367)
  MoveL 7816 to (-41.16, 146.07, 116.27) mm, rotated rx 180 ry 0 rz 180 deg; joints [-144.015, 69.718, -81.193, 143.463, 80.736, 6.802]
  MoveL 7817 to (-41.16, 146.07, 116.27) mm, rotated rx 180 ry 0 rz 180 deg; joints [-144.015, 69.718, -81.193, 143.463, 80.736, 6.802]
  Call Extruder(12.35641)
  MoveL 7818 to (-41.2, 145.48, 116.27) mm, rotated rx 180 ry 0 rz 180 deg; joints [-144.131, 69.698, -81.213, 143.576, 80.69, 6.807]
  MoveL 7819 to (-41.2, 145.48, 116.27) mm, rotated rx 180 ry 0 rz 180 deg; joints [-144.131, 69.698, -81.213, 143.576, 80.69, 6.807]
  Call Extruder(12.92986)
  MoveL 7820 to (-41.25, 144.32, 116.27) mm, rotated rx -180 ry 0 rz -180 deg; joints [-144.355, 69.657, -81.255, 143.794, 80.597, 6.821]
  MoveL 7821 to (-41.25, 144.32, 116.27) mm, rotated rx -180 ry 0 rz -180 deg; joints [-144.355, 69.657, -81.255, 143.794, 80.597, 6.821]
  Call Extruder(13.64382)
  MoveL 7822 to (-41.29, 142.86, 116.27) mm, rotated rx -180 ry 0 rz 180 deg; joints [-144.635, 69.604, -81.308, 144.065, 80.478, 6.837]
  Call Extruder(55.70865)
  MoveL 7823 to (-41.29, 57.14, 116.27) mm, rotated rx -180 ry 0 rz 180 deg; joints [-164.153, 66.947, -83.493, 163.505, 74.1, 4.638]
  Call Extruder(56.13720)
  MoveL 7824 to (-41.27, 56.26, 116.27) mm, rotated rx 180 ry 0 rz 180 deg; joints [-164.382, 66.928, -83.506, 163.74, 74.05, 4.582]
  MoveL 7825 to (-41.27, 56.26, 116.27) mm, rotated rx 180 ry 0 rz 180 deg; joints [-164.382, 66.928, -83.506, 163.74, 74.05, 4.582]
  Call Extruder(56.71065)
  MoveL 7826 to (-41.23, 55.1, 116.27) mm, rotated rx -180 ry 0 rz -180 deg; joints [-164.686, 66.9, -83.524, 164.051, 73.983, 4.509]
  MoveL 7827 to (-41.23, 55.1, 116.27) mm, rotated rx -180 ry 0 rz -180 deg; joints [-164.686, 66.9, -83.524, 164.051, 73.983, 4.509]
  Call Extruder(57.14497)
  MoveL 7828 to (-41.18, 54.23, 116.27) mm, rotated rx -180 ry 0 rz -180 deg; joints [-164.915, 66.879, -83.538, 164.286, 73.931, 4.453]
  MoveL 7829 to (-41.18, 54.23, 116.27) mm, rotated rx -180 ry 0 rz -180 deg; joints [-164.915, 66.879, -83.538, 164.286, 73.931, 4.453]
  Call Extruder(57.43904)
  MoveL 7830 to (-41.13, 53.64, 116.27) mm, rotated rx 180 ry 0 rz -180 deg; joints [-165.068, 66.864, -83.548, 164.443, 73.895, 4.416]
  MoveL 7831 to (-41.13, 53.64, 116.27) mm, rotated rx 180 ry 0 rz -180 deg; joints [-165.068, 66.864, -83.548, 164.443, 73.895, 4.416]
  Call Extruder(57.73444)
  MoveL 7832 to (-41.09, 53.05, 116.27) mm, rotated rx -180 ry 0 rz -180 deg; joints [-165.222, 66.849, -83.558, 164.601, 73.859, 4.379]
  MoveL 7833 to (-41.09, 53.05, 116.27) mm, rotated rx -180 ry 0 rz -180 deg; joints [-165.222, 66.849, -83.558, 164.601, 73.859, 4.379]
  Call Extruder(57.98067)
  MoveL 7834 to (-41.04, 52.56, 116.27) mm, rotated rx -180 ry 0 rz -180 deg; joints [-165.349, 66.836, -83.566, 164.731, 73.829, 4.348]
  MoveL 7835 to (-41.04, 52.56, 116.27) mm, rotated rx -180 ry 0 rz -180 deg; joints [-165.349, 66.836, -83.566, 164.731, 73.829, 4.348]
  Call Extruder(58.17738)
  MoveL 7836 to (-40.99, 52.17, 116.27) mm, rotated rx -180 ry 0 rz -180 deg; joints [-165.449, 66.825, -83.574, 164.834, 73.804, 4.324]
  MoveL 7837 to (-40.99, 52.17, 116.27) mm, rotated rx -180 ry 0 rz -180 deg; joints [-165.449, 66.825, -83.574, 164.834, 73.804, 4.324]
  Call Extruder(58.37495)
  MoveL 7838 to (-40.95, 51.78, 116.27) mm, rotated rx -180 ry 0 rz 180 deg; joints [-165.549, 66.814, -83.581, 164.936, 73.779, 4.3]
  MoveL 7839 to (-40.95, 51.78, 116.27) mm, rotated rx -180 ry 0 rz 180 deg; joints [-165.549, 66.814, -83.581, 164.936, 73.779, 4.3]
  Call Extruder(58.57339)
  MoveL 7840 to (-40.9, 51.4, 116.27) mm, rotated rx -180 ry 0 rz -180 deg; joints [-165.65, 66.803, -83.588, 165.04, 73.754, 4.275]
  MoveL 7841 to (-40.9, 51.4, 116.27) mm, rotated rx -180 ry 0 rz -180 deg; joints [-165.65, 66.803, -83.588, 165.04, 73.754, 4.275]
  Call Extruder(58.77270)
  MoveL 7842 to (-40.86, 51.01, 116.27) mm, rotated rx -180 ry 0 rz 180 deg; joints [-165.751, 66.792, -83.595, 165.143, 73.729, 4.251]
  MoveL 7843 to (-40.86, 51.01, 116.27) mm, rotated rx -180 ry 0 rz 180 deg; joints [-165.751, 66.792, -83.595, 165.143, 73.729, 4.251]
  Call Extruder(58.93152)
  MoveL 7844 to (-40.81, 50.7, 116.27) mm, rotated rx -180 ry 0 rz -180 deg; joints [-165.829, 66.783, -83.601, 165.223, 73.708, 4.232]
  MoveL 7845 to (-40.81, 50.7, 116.27) mm, rotated rx -180 ry 0 rz -180 deg; joints [-165.829, 66.783, -83.601, 165.223, 73.708, 4.232]
  Call Extruder(59.09106)
  MoveL 7846 to (-40.76, 50.4, 116.27) mm, rotated rx 180 ry 0 rz 180 deg; joints [-165.908, 66.773, -83.607, 165.304, 73.687, 4.213]
  MoveL 7847 to (-40.76, 50.4, 116.27) mm, rotated rx 180 ry 0 rz 180 deg; joints [-165.908, 66.773, -83.607, 165.304, 73.687, 4.213]
  Call Extruder(59.25133)
  MoveL 7848 to (-40.71, 50.09, 116.27) mm, rotated rx -180 ry 0 rz -180 deg; joints [-165.987, 66.764, -83.613, 165.385, 73.667, 4.194]
  MoveL 7849 to (-40.71, 50.09, 116.27) mm, rotated rx -180 ry 0 rz -180 deg; joints [-165.987, 66.764, -83.613, 165.385, 73.667, 4.194]
  Call Extruder(59.41232)
  MoveL 7850 to (-40.66, 49.79, 116.27) mm, rotated rx -180 ry 0 rz 180 deg; joints [-166.066, 66.755, -83.619, 165.466, 73.646, 4.175]
  MoveL 7851 to (-40.66, 49.79, 116.27) mm, rotated rx -180 ry 0 rz 180 deg; joints [-166.066, 66.755, -83.619, 165.466, 73.646, 4.175]
  Call Extruder(59.57405)
  MoveL 7852 to (-40.61, 49.48, 116.27) mm, rotated rx 180 ry 0 rz 180 deg; joints [-166.145, 66.745, -83.625, 165.547, 73.625, 4.156]
  MoveL 7853 to (-40.61, 49.48, 116.27) mm, rotated rx 180 ry 0 rz 180 deg; joints [-166.145, 66.745, -83.625, 165.547, 73.625, 4.156]
  Call Extruder(59.73650)
  MoveL 7854 to (-40.56, 49.17, 116.27) mm, rotated rx -180 ry 0 rz -180 deg; joints [-166.224, 66.736, -83.631, 165.628, 73.605, 4.137]
  MoveL 7855 to (-40.56, 49.17, 116.27) mm, rotated rx -180 ry 0 rz -180 deg; joints [-166.224, 66.736, -83.631, 165.628, 73.605, 4.137]
  Call Extruder(59.87043)
  MoveL 7856 to (-40.52, 48.93, 116.27) mm, rotated rx -180 ry 0 rz -180 deg; joints [-166.288, 66.728, -83.637, 165.693, 73.587, 4.122]
  MoveL 7857 to (-40.52, 48.93, 116.27) mm, rotated rx -180 ry 0 rz -180 deg; joints [-166.288, 66.728, -83.637, 165.693, 73.587, 4.122]
  Call Extruder(60.00496)
  MoveL 7858 to (-40.47, 48.68, 116.27) mm, rotated rx -180 ry 0 rz -180 deg; joints [-166.352, 66.719, -83.642, 165.759, 73.569, 4.106]
  MoveL 7859 to (-40.47, 48.68, 116.27) mm, rotated rx -180 ry 0 rz -180 deg; joints [-166.352, 66.719, -83.642, 165.759, 73.569, 4.106]
  Call Extruder(60.14011)
  MoveL 7860 to (-40.42, 48.43, 116.27) mm, rotated rx 180 ry 0 rz 180 deg; joints [-166.416, 66.711, -83.647, 165.824, 73.551, 4.091]
  MoveL 7861 to (-40.42, 48.43, 116.27) mm, rotated rx 180 ry 0 rz 180 deg; joints [-166.416, 66.711, -83.647, 165.824, 73.551, 4.091]
  Call Extruder(60.27586)
  MoveL 7862 to (-40.37, 48.18, 116.27) mm, rotated rx -180 ry 0 rz 180 deg; joints [-166.48, 66.703, -83.653, 165.89, 73.533, 4.076]
  MoveL 7863 to (-40.37, 48.18, 116.27) mm, rotated rx -180 ry 0 rz 180 deg; joints [-166.48, 66.703, -83.653, 165.89, 73.533, 4.076]
  Call Extruder(60.41223)
  MoveL 7864 to (-40.32, 47.93, 116.27) mm, rotated rx -180 ry 0 rz -180 deg; joints [-166.544, 66.695, -83.658, 165.956, 73.516, 4.06]
  MoveL 7865 to (-40.32, 47.93, 116.27) mm, rotated rx -180 ry 0 rz -180 deg; joints [-166.544, 66.695, -83.658, 165.956, 73.516, 4.06]
  Call Extruder(60.54920)
  MoveL 7866 to (-40.27, 47.68, 116.27) mm, rotated rx 180 ry 0 rz -180 deg; joints [-166.608, 66.686, -83.663, 166.022, 73.498, 4.045]
  MoveL 7867 to (-40.27, 47.68, 116.27) mm, rotated rx 180 ry 0 rz -180 deg; joints [-166.608, 66.686, -83.663, 166.022, 73.498, 4.045]
  Call Extruder(60.68679)
  MoveL 7868 to (-40.22, 47.43, 116.27) mm, rotated rx 180 ry 0 rz 180 deg; joints [-166.673, 66.678, -83.669, 166.087, 73.48, 4.029]
  MoveL 7869 to (-40.22, 47.43, 116.27) mm, rotated rx 180 ry 0 rz 180 deg; joints [-166.673, 66.678, -83.669, 166.087, 73.48, 4.029]
  Call Extruder(60.80052)
  MoveL 7870 to (-40.17, 47.23, 116.27) mm, rotated rx 180 ry 0 rz -180 deg; joints [-166.725, 66.671, -83.673, 166.141, 73.466, 4.016]
  MoveL 7871 to (-40.17, 47.23, 116.27) mm, rotated rx 180 ry 0 rz -180 deg; joints [-166.725, 66.671, -83.673, 166.141, 73.466, 4.016]
  Call Extruder(60.91470)
  MoveL 7872 to (-40.13, 47.02, 116.27) mm, rotated rx -180 ry 0 rz 180 deg; joints [-166.778, 66.664, -83.678, 166.195, 73.451, 4.004]
  MoveL 7873 to (-40.13, 47.02, 116.27) mm, rotated rx -180 ry 0 rz 180 deg; joints [-166.778, 66.664, -83.678, 166.195, 73.451, 4.004]
  Call Extruder(61.02933)
  MoveL 7874 to (-40.08, 46.82, 116.27) mm, rotated rx 180 ry 0 rz -180 deg; joints [-166.83, 66.657, -83.682, 166.249, 73.436, 3.991]
  MoveL 7875 to (-40.08, 46.82, 116.27) mm, rotated rx 180 ry 0 rz -180 deg; joints [-166.83, 66.657, -83.682, 166.249, 73.436, 3.991]
  Call Extruder(61.14442)
  MoveL 7876 to (-40.04, 46.61, 116.27) mm, rotated rx -180 ry 0 rz -180 deg; joints [-166.883, 66.65, -83.687, 166.303, 73.421, 3.978]
  MoveL 7877 to (-40.04, 46.61, 116.27) mm, rotated rx -180 ry 0 rz -180 deg; joints [-166.883, 66.65, -83.687, 166.303, 73.421, 3.978]
  Call Extruder(61.26666)
  MoveL 7878 to (-39.98, 46.4, 116.27) mm, rotated rx -180 ry 0 rz -180 deg; joints [-166.937, 66.642, -83.692, 166.359, 73.405, 3.965]
  MoveL 7879 to (-39.98, 46.4, 116.27) mm, rotated rx -180 ry 0 rz -180 deg; joints [-166.937, 66.642, -83.692, 166.359, 73.405, 3.965]
  Call Extruder(61.39632)
  MoveL 7880 to (-39.92, 46.18, 116.27) mm, rotated rx 180 ry 0 rz 180 deg; joints [-166.994, 66.633, -83.697, 166.417, 73.386, 3.952]
  MoveL 7881 to (-39.92, 46.18, 116.27) mm, rotated rx 180 ry 0 rz 180 deg; joints [-166.994, 66.633, -83.697, 166.417, 73.386, 3.952]
  Call Extruder(61.52655)
  MoveL 7882 to (-39.85, 45.95, 116.27) mm, rotated rx -180 ry 0 rz -180 deg; joints [-167.051, 66.624, -83.703, 166.475, 73.368, 3.939]
  MoveL 7883 to (-39.85, 45.95, 116.27) mm, rotated rx -180 ry 0 rz -180 deg; joints [-167.051, 66.624, -83.703, 166.475, 73.368, 3.939]
  Call Extruder(61.65735)
  MoveL 7884 to (-39.78, 45.73, 116.27) mm, rotated rx 180 ry 0 rz 180 deg; joints [-167.107, 66.615, -83.709, 166.533, 73.35, 3.925]
  MoveL 7885 to (-39.78, 45.73, 116.27) mm, rotated rx 180 ry 0 rz 180 deg; joints [-167.107, 66.615, -83.709, 166.533, 73.35, 3.925]
  Call Extruder(61.78871)
  MoveL 7886 to (-39.71, 45.5, 116.27) mm, rotated rx -180 ry 0 rz -180 deg; joints [-167.164, 66.606, -83.715, 166.591, 73.331, 3.912]
  MoveL 7887 to (-39.71, 45.5, 116.27) mm, rotated rx -180 ry 0 rz -180 deg; joints [-167.164, 66.606, -83.715, 166.591, 73.331, 3.912]
  Call Extruder(61.90061)
  MoveL 7888 to (-39.65, 45.32, 116.27) mm, rotated rx 180 ry 0 rz 180 deg; joints [-167.212, 66.598, -83.72, 166.639, 73.316, 3.901]
  MoveL 7889 to (-39.65, 45.32, 116.27) mm, rotated rx 180 ry 0 rz 180 deg; joints [-167.212, 66.598, -83.72, 166.639, 73.316, 3.901]
  Call Extruder(62.01295)
  MoveL 7890 to (-39.59, 45.13, 116.27) mm, rotated rx 180 ry 0 rz -180 deg; joints [-167.26, 66.59, -83.725, 166.688, 73.3, 3.89]
  MoveL 7891 to (-39.59, 45.13, 116.27) mm, rotated rx 180 ry 0 rz -180 deg; joints [-167.26, 66.59, -83.725, 166.688, 73.3, 3.89]
  Call Extruder(62.12574)
  MoveL 7892 to (-39.53, 44.94, 116.27) mm, rotated rx 180 ry 0 rz 180 deg; joints [-167.307, 66.582, -83.73, 166.737, 73.284, 3.879]
  MoveL 7893 to (-39.53, 44.94, 116.27) mm, rotated rx 180 ry 0 rz 180 deg; joints [-167.307, 66.582, -83.73, 166.737, 73.284, 3.879]
  Call Extruder(62.23898)
  MoveL 7894 to (-39.47, 44.75, 116.27) mm, rotated rx -180 ry 0 rz 180 deg; joints [-167.355, 66.574, -83.735, 166.786, 73.268, 3.867]
  MoveL 7895 to (-39.47, 44.75, 116.27) mm, rotated rx -180 ry 0 rz 180 deg; joints [-167.355, 66.574, -83.735, 166.786, 73.268, 3.867]
  Call Extruder(62.35266)
  MoveL 7896 to (-39.41, 44.56, 116.27) mm, rotated rx 180 ry 0 rz -180 deg; joints [-167.403, 66.566, -83.74, 166.835, 73.252, 3.856]
  MoveL 7897 to (-39.41, 44.56, 116.27) mm, rotated rx 180 ry 0 rz -180 deg; joints [-167.403, 66.566, -83.74, 166.835, 73.252, 3.856]
  Call Extruder(62.53462)
  MoveL 7898 to (-39.29, 44.27, 116.27) mm, rotated rx -180 ry 0 rz 180 deg; joints [-167.475, 66.552, -83.749, 166.909, 73.225, 3.84]
  MoveL 7899 to (-39.29, 44.27, 116.27) mm, rotated rx -180 ry 0 rz 180 deg; joints [-167.475, 66.552, -83.749, 166.909, 73.225, 3.84]
  Call Extruder(62.71734)
  MoveL 7900 to (-39.17, 43.98, 116.27) mm, rotated rx -180 ry 0 rz 180 deg; joints [-167.548, 66.538, -83.757, 166.983, 73.198, 3.823]
  MoveL 7901 to (-39.17, 43.98, 116.27) mm, rotated rx -180 ry 0 rz 180 deg; joints [-167.548, 66.538, -83.757, 166.983, 73.198, 3.823]
  Call Extruder(62.88775)
  MoveL 7902 to (-39.05, 43.71, 116.27) mm, rotated rx -180 ry 0 rz -180 deg; joints [-167.615, 66.525, -83.766, 167.052, 73.172, 3.808]
  MoveL 7903 to (-39.05, 43.71, 116.27) mm, rotated rx -180 ry 0 rz -180 deg; joints [-167.615, 66.525, -83.766, 167.052, 73.172, 3.808]
  Call Extruder(63.04573)
  MoveL 7904 to (-38.94, 43.46, 116.27) mm, rotated rx 180 ry 0 rz -180 deg; joints [-167.677, 66.512, -83.773, 167.115, 73.148, 3.794]
  MoveL 7905 to (-38.94, 43.46, 116.27) mm, rotated rx 180 ry 0 rz -180 deg; joints [-167.677, 66.512, -83.773, 167.115, 73.148, 3.794]
  Call Extruder(63.20432)
  MoveL 7906 to (-38.84, 43.21, 116.27) mm, rotated rx -180 ry 0 rz 180 deg; joints [-167.739, 66.5, -83.781, 167.179, 73.125, 3.78]
  MoveL 7907 to (-38.84, 43.21, 116.27) mm, rotated rx -180 ry 0 rz 180 deg; joints [-167.739, 66.5, -83.781, 167.179, 73.125, 3.78]
  Call Extruder(63.41049)
  MoveL 7908 to (-38.66, 42.91, 116.27) mm, rotated rx 180 ry 0 rz -180 deg; joints [-167.813, 66.481, -83.793, 167.253, 73.091, 3.765]
  MoveL 7909 to (-38.66, 42.91, 116.27) mm, rotated rx 180 ry 0 rz -180 deg; joints [-167.813, 66.481, -83.793, 167.253, 73.091, 3.765]
  Call Extruder(63.61743)
  MoveL 7910 to (-38.49, 42.6, 116.27) mm, rotated rx 180 ry 0 rz 180 deg; joints [-167.886, 66.463, -83.804, 167.327, 73.056, 3.749]
  MoveL 7911 to (-38.49, 42.6, 116.27) mm, rotated rx 180 ry 0 rz 180 deg; joints [-167.886, 66.463, -83.804, 167.327, 73.056, 3.749]
  Call Extruder(63.82516)
  MoveL 7912 to (-38.31, 42.3, 116.27) mm, rotated rx 180 ry 0 rz 180 deg; joints [-167.96, 66.444, -83.816, 167.402, 73.023, 3.734]
  MoveL 7913 to (-38.31, 42.3, 116.27) mm, rotated rx 180 ry 0 rz 180 deg; joints [-167.96, 66.444, -83.816, 167.402, 73.023, 3.734]
  Call Extruder(64.03366)
  MoveL 7914 to (-38.14, 41.99, 116.27) mm, rotated rx -180 ry 0 rz -180 deg; joints [-168.033, 66.426, -83.827, 167.477, 72.988, 3.718]
  MoveL 7915 to (-38.14, 41.99, 116.27) mm, rotated rx -180 ry 0 rz -180 deg; joints [-168.033, 66.426, -83.827, 167.477, 72.988, 3.718]
  Call Extruder(64.21320)
  MoveL 7916 to (-37.96, 41.75, 116.27) mm, rotated rx 180 ry 0 rz -180 deg; joints [-168.091, 66.408, -83.838, 167.535, 72.957, 3.707]
  MoveL 7917 to (-37.96, 41.75, 116.27) mm, rotated rx 180 ry 0 rz -180 deg; joints [-168.091, 66.408, -83.838, 167.535, 72.957, 3.707]
  Call Extruder(64.54664)
  MoveL 7918 to (-37.63, 41.3, 116.27) mm, rotated rx -180 ry 0 rz -180 deg; joints [-168.197, 66.375, -83.858, 167.643, 72.899, 3.686]
  MoveL 7919 to (-37.63, 41.3, 116.27) mm, rotated rx -180 ry 0 rz -180 deg; joints [-168.197, 66.375, -83.858, 167.643, 72.899, 3.686]
  Call Extruder(64.88126)
  MoveL 7920 to (-37.3, 40.85, 116.27) mm, rotated rx 180 ry 0 rz 180 deg; joints [-168.304, 66.343, -83.878, 167.751, 72.841, 3.665]
  Call Extruder(65.70919)
  MoveL 7921 to (-36.39, 39.81, 116.27) mm, rotated rx -180 ry 0 rz 180 deg; joints [-168.541, 66.255, -83.931, 167.99, 72.688, 3.622]
  Call Extruder(66.53710)
  MoveL 7922 to (-35.35, 38.9, 116.27) mm, rotated rx -180 ry 0 rz -180 deg; joints [-168.739, 66.16, -83.988, 168.187, 72.527, 3.593]
  Call Extruder(66.70441)
  MoveL 7923 to (-35.13, 38.73, 116.27) mm, rotated rx -180 ry 0 rz 180 deg; joints [-168.773, 66.14, -83.999, 168.22, 72.493, 3.59]
  MoveL 7924 to (-35.13, 38.73, 116.27) mm, rotated rx -180 ry 0 rz 180 deg; joints [-168.773, 66.14, -83.999, 168.22, 72.493, 3.59]
  Call Extruder(67.03783)
  MoveL 7925 to (-34.68, 38.4, 116.27) mm, rotated rx -180 ry 0 rz 180 deg; joints [-168.84, 66.099, -84.023, 168.286, 72.426, 3.582]
  MoveL 7926 to (-34.68, 38.4, 116.27) mm, rotated rx -180 ry 0 rz 180 deg; joints [-168.84, 66.099, -84.023, 168.286, 72.426, 3.582]
  Call Extruder(67.37007)
  MoveL 7927 to (-34.23, 38.08, 116.27) mm, rotated rx -180 ry 0 rz -180 deg; joints [-168.908, 66.059, -84.047, 168.354, 72.359, 3.574]
  MoveL 7928 to (-34.23, 38.08, 116.27) mm, rotated rx -180 ry 0 rz -180 deg; joints [-168.908, 66.059, -84.047, 168.354, 72.359, 3.574]
  Call Extruder(67.48778)
  MoveL 7929 to (-34.05, 37.98, 116.27) mm, rotated rx -180 ry 0 rz 180 deg; joints [-168.927, 66.044, -84.056, 168.372, 72.334, 3.573]
  MoveL 7930 to (-34.05, 37.98, 116.27) mm, rotated rx -180 ry 0 rz 180 deg; joints [-168.927, 66.044, -84.056, 168.372, 72.334, 3.573]
  Call Extruder(67.69550)
  MoveL 7931 to (-33.75, 37.8, 116.27) mm, rotated rx -180 ry 0 rz 180 deg; joints [-168.96, 66.017, -84.071, 168.404, 72.291, 3.572]
  MoveL 7932 to (-33.75, 37.8, 116.27) mm, rotated rx -180 ry 0 rz 180 deg; joints [-168.96, 66.017, -84.071, 168.404, 72.291, 3.572]
  Call Extruder(67.90244)
  MoveL 7933 to (-33.45, 37.63, 116.27) mm, rotated rx 180 ry 0 rz 180 deg; joints [-168.993, 65.99, -84.087, 168.435, 72.248, 3.57]
  MoveL 7934 to (-33.45, 37.63, 116.27) mm, rotated rx 180 ry 0 rz 180 deg; joints [-168.993, 65.99, -84.087, 168.435, 72.248, 3.57]
  Call Extruder(68.10860)
  MoveL 7935 to (-33.14, 37.45, 116.27) mm, rotated rx -180 ry 0 rz -180 deg; joints [-169.026, 65.964, -84.102, 168.467, 72.204, 3.568]
  MoveL 7936 to (-33.14, 37.45, 116.27) mm, rotated rx -180 ry 0 rz -180 deg; joints [-169.026, 65.964, -84.102, 168.467, 72.204, 3.568]
  Call Extruder(68.29029)
  MoveL 7937 to (-32.86, 37.31, 116.27) mm, rotated rx -180 ry 0 rz -180 deg; joints [-169.052, 65.94, -84.116, 168.492, 72.166, 3.568]
  MoveL 7938 to (-32.86, 37.31, 116.27) mm, rotated rx -180 ry 0 rz -180 deg; joints [-169.052, 65.94, -84.116, 168.492, 72.166, 3.568]
  Call Extruder(68.44829)
  MoveL 7939 to (-32.62, 37.2, 116.27) mm, rotated rx -180 ry 0 rz 180 deg; joints [-169.068, 65.918, -84.128, 168.507, 72.132, 3.57]
  MoveL 7940 to (-32.62, 37.2, 116.27) mm, rotated rx -180 ry 0 rz 180 deg; joints [-169.068, 65.918, -84.128, 168.507, 72.132, 3.57]
  Call Extruder(68.60569)
  MoveL 7941 to (-32.37, 37.09, 116.27) mm, rotated rx 180 ry 0 rz 180 deg; joints [-169.085, 65.897, -84.141, 168.523, 72.098, 3.571]
  MoveL 7942 to (-32.37, 37.09, 116.27) mm, rotated rx 180 ry 0 rz 180 deg; joints [-169.085, 65.897, -84.141, 168.523, 72.098, 3.571]
  Call Extruder(68.78840)
  MoveL 7943 to (-32.08, 36.97, 116.27) mm, rotated rx -180 ry 0 rz 180 deg; joints [-169.104, 65.872, -84.155, 168.539, 72.058, 3.574]
  MoveL 7944 to (-32.08, 36.97, 116.27) mm, rotated rx -180 ry 0 rz 180 deg; joints [-169.104, 65.872, -84.155, 168.539, 72.058, 3.574]
  Call Extruder(68.97035)
  MoveL 7945 to (-31.78, 36.85, 116.27) mm, rotated rx -180 ry 0 rz -180 deg; joints [-169.122, 65.847, -84.169, 168.556, 72.018, 3.576]
  MoveL 7946 to (-31.78, 36.85, 116.27) mm, rotated rx -180 ry 0 rz -180 deg; joints [-169.122, 65.847, -84.169, 168.556, 72.018, 3.576]
  Call Extruder(69.11768)
  MoveL 7947 to (-31.54, 36.76, 116.27) mm, rotated rx -180 ry 0 rz -180 deg; joints [-169.135, 65.826, -84.181, 168.568, 71.986, 3.578]
  MoveL 7948 to (-31.54, 36.76, 116.27) mm, rotated rx -180 ry 0 rz -180 deg; joints [-169.135, 65.826, -84.181, 168.568, 71.986, 3.578]
  Call Extruder(69.23091)
  MoveL 7949 to (-31.35, 36.7, 116.27) mm, rotated rx 180 ry 0 rz 180 deg; joints [-169.143, 65.81, -84.19, 168.574, 71.961, 3.581]
  MoveL 7950 to (-31.35, 36.7, 116.27) mm, rotated rx 180 ry 0 rz 180 deg; joints [-169.143, 65.81, -84.19, 168.574, 71.961, 3.581]
  Call Extruder(69.34371)
  MoveL 7951 to (-31.17, 36.64, 116.27) mm, rotated rx 180 ry 0 rz 180 deg; joints [-169.15, 65.794, -84.198, 168.58, 71.936, 3.584]
  MoveL 7952 to (-31.17, 36.64, 116.27) mm, rotated rx 180 ry 0 rz 180 deg; joints [-169.15, 65.794, -84.198, 168.58, 71.936, 3.584]
  Call Extruder(69.45605)
  MoveL 7953 to (-30.98, 36.58, 116.27) mm, rotated rx -180 ry 0 rz 180 deg; joints [-169.157, 65.778, -84.207, 168.586, 71.911, 3.587]
  MoveL 7954 to (-30.98, 36.58, 116.27) mm, rotated rx -180 ry 0 rz 180 deg; joints [-169.157, 65.778, -84.207, 168.586, 71.911, 3.587]
  Call Extruder(69.56796)
  MoveL 7955 to (-30.79, 36.52, 116.27) mm, rotated rx -180 ry 0 rz 180 deg; joints [-169.164, 65.762, -84.216, 168.592, 71.886, 3.59]
  MoveL 7956 to (-30.79, 36.52, 116.27) mm, rotated rx -180 ry 0 rz 180 deg; joints [-169.164, 65.762, -84.216, 168.592, 71.886, 3.59]
  Call Extruder(69.68936)
  MoveL 7957 to (-30.58, 36.45, 116.27) mm, rotated rx 180 ry 0 rz 180 deg; joints [-169.172, 65.745, -84.226, 168.598, 71.859, 3.593]
  MoveL 7958 to (-30.58, 36.45, 116.27) mm, rotated rx 180 ry 0 rz 180 deg; joints [-169.172, 65.745, -84.226, 168.598, 71.859, 3.593]
  Call Extruder(69.82015)
  MoveL 7959 to (-30.36, 36.38, 116.27) mm, rotated rx -180 ry 0 rz 180 deg; joints [-169.179, 65.726, -84.237, 168.604, 71.83, 3.597]
  MoveL 7960 to (-30.36, 36.38, 116.27) mm, rotated rx -180 ry 0 rz 180 deg; joints [-169.179, 65.726, -84.237, 168.604, 71.83, 3.597]
  Call Extruder(69.95037)
  MoveL 7961 to (-30.14, 36.32, 116.27) mm, rotated rx 180 ry 0 rz -180 deg; joints [-169.186, 65.707, -84.247, 168.609, 71.801, 3.6]
  MoveL 7962 to (-30.14, 36.32, 116.27) mm, rotated rx 180 ry 0 rz -180 deg; joints [-169.186, 65.707, -84.247, 168.609, 71.801, 3.6]
  Call Extruder(70.08003)
  MoveL 7963 to (-29.91, 36.25, 116.27) mm, rotated rx -180 ry 0 rz -180 deg; joints [-169.193, 65.688, -84.258, 168.615, 71.771, 3.604]
  MoveL 7964 to (-29.91, 36.25, 116.27) mm, rotated rx -180 ry 0 rz -180 deg; joints [-169.193, 65.688, -84.258, 168.615, 71.771, 3.604]
  Call Extruder(70.20913)
  MoveL 7965 to (-29.69, 36.18, 116.27) mm, rotated rx -180 ry 0 rz -180 deg; joints [-169.201, 65.669, -84.268, 168.621, 71.742, 3.608]
  MoveL 7966 to (-29.69, 36.18, 116.27) mm, rotated rx -180 ry 0 rz -180 deg; joints [-169.201, 65.669, -84.268, 168.621, 71.742, 3.608]
  Call Extruder(70.32420)
  MoveL 7967 to (-29.48, 36.14, 116.27) mm, rotated rx -180 ry 0 rz 180 deg; joints [-169.202, 65.652, -84.278, 168.621, 71.716, 3.613]
  MoveL 7968 to (-29.48, 36.14, 116.27) mm, rotated rx -180 ry 0 rz 180 deg; joints [-169.202, 65.652, -84.278, 168.621, 71.716, 3.613]
  Call Extruder(70.43882)
  MoveL 7969 to (-29.28, 36.09, 116.27) mm, rotated rx -180 ry 0 rz -180 deg; joints [-169.204, 65.635, -84.287, 168.621, 71.69, 3.618]
  MoveL 7970 to (-29.28, 36.09, 116.27) mm, rotated rx -180 ry 0 rz -180 deg; joints [-169.204, 65.635, -84.287, 168.621, 71.69, 3.618]
  Call Extruder(70.55299)
  MoveL 7971 to (-29.08, 36.05, 116.27) mm, rotated rx -180 ry 0 rz 180 deg; joints [-169.206, 65.618, -84.296, 168.621, 71.664, 3.623]
  MoveL 7972 to (-29.08, 36.05, 116.27) mm, rotated rx -180 ry 0 rz 180 deg; joints [-169.206, 65.618, -84.296, 168.621, 71.664, 3.623]
  Call Extruder(70.66671)
  MoveL 7973 to (-28.87, 36, 116.27) mm, rotated rx 180 ry 0 rz 180 deg; joints [-169.207, 65.601, -84.306, 168.621, 71.638, 3.628]
  MoveL 7974 to (-28.87, 36, 116.27) mm, rotated rx 180 ry 0 rz 180 deg; joints [-169.207, 65.601, -84.306, 168.621, 71.638, 3.628]
  Call Extruder(70.79213)
  MoveL 7975 to (-28.65, 35.96, 116.27) mm, rotated rx 180 ry 0 rz 180 deg; joints [-169.208, 65.582, -84.316, 168.62, 71.609, 3.633]
  MoveL 7976 to (-28.65, 35.96, 116.27) mm, rotated rx 180 ry 0 rz 180 deg; joints [-169.208, 65.582, -84.316, 168.62, 71.609, 3.633]
  Call Extruder(70.92911)
  MoveL 7977 to (-28.4, 35.91, 116.27) mm, rotated rx -180 ry 0 rz 180 deg; joints [-169.209, 65.561, -84.327, 168.619, 71.577, 3.64]
  MoveL 7978 to (-28.4, 35.91, 116.27) mm, rotated rx -180 ry 0 rz 180 deg; joints [-169.209, 65.561, -84.327, 168.619, 71.577, 3.64]
  Call Extruder(71.06547)
  MoveL 7979 to (-28.15, 35.86, 116.27) mm, rotated rx 180 ry 0 rz 180 deg; joints [-169.21, 65.54, -84.339, 168.617, 71.546, 3.646]
  MoveL 7980 to (-28.15, 35.86, 116.27) mm, rotated rx 180 ry 0 rz 180 deg; joints [-169.21, 65.54, -84.339, 168.617, 71.546, 3.646]
  Call Extruder(71.20123)
  MoveL 7981 to (-27.9, 35.81, 116.27) mm, rotated rx 180 ry 0 rz 180 deg; joints [-169.21, 65.519, -84.35, 168.616, 71.514, 3.653]
  MoveL 7982 to (-27.9, 35.81, 116.27) mm, rotated rx 180 ry 0 rz 180 deg; joints [-169.21, 65.519, -84.35, 168.616, 71.514, 3.653]
  Call Extruder(71.33638)
  MoveL 7983 to (-27.65, 35.76, 116.27) mm, rotated rx 180 ry 0 rz 180 deg; joints [-169.211, 65.498, -84.361, 168.614, 71.483, 3.659]
  MoveL 7984 to (-27.65, 35.76, 116.27) mm, rotated rx 180 ry 0 rz 180 deg; joints [-169.211, 65.498, -84.361, 168.614, 71.483, 3.659]
  Call Extruder(71.47091)
  MoveL 7985 to (-27.4, 35.71, 116.27) mm, rotated rx 180 ry 0 rz -180 deg; joints [-169.212, 65.477, -84.372, 168.613, 71.451, 3.666]
  MoveL 7986 to (-27.4, 35.71, 116.27) mm, rotated rx 180 ry 0 rz -180 deg; joints [-169.212, 65.477, -84.372, 168.613, 71.451, 3.666]
  Call Extruder(71.60484)
  MoveL 7987 to (-27.15, 35.66, 116.27) mm, rotated rx -180 ry 0 rz -180 deg; joints [-169.212, 65.456, -84.383, 168.611, 71.42, 3.672]
  MoveL 7988 to (-27.15, 35.66, 116.27) mm, rotated rx -180 ry 0 rz -180 deg; joints [-169.212, 65.456, -84.383, 168.611, 71.42, 3.672]
  Call Extruder(71.75270)
  MoveL 7989 to (-26.87, 35.61, 116.27) mm, rotated rx -180 ry 0 rz -180 deg; joints [-169.211, 65.433, -84.396, 168.608, 71.385, 3.68]
  MoveL 7990 to (-26.87, 35.61, 116.27) mm, rotated rx -180 ry 0 rz -180 deg; joints [-169.211, 65.433, -84.396, 168.608, 71.385, 3.68]
  Call Extruder(71.91443)
  MoveL 7991 to (-26.57, 35.56, 116.27) mm, rotated rx 180 ry 0 rz -180 deg; joints [-169.208, 65.407, -84.409, 168.602, 71.347, 3.689]
  MoveL 7992 to (-26.57, 35.56, 116.27) mm, rotated rx 180 ry 0 rz -180 deg; joints [-169.208, 65.407, -84.409, 168.602, 71.347, 3.689]
  Call Extruder(72.07544)
  MoveL 7993 to (-26.26, 35.51, 116.27) mm, rotated rx 180 ry 0 rz -180 deg; joints [-169.205, 65.382, -84.423, 168.596, 71.308, 3.699]
  MoveL 7994 to (-26.26, 35.51, 116.27) mm, rotated rx 180 ry 0 rz -180 deg; joints [-169.205, 65.382, -84.423, 168.596, 71.308, 3.699]
  Call Extruder(72.23572)
  MoveL 7995 to (-25.96, 35.46, 116.27) mm, rotated rx -180 ry 0 rz 180 deg; joints [-169.202, 65.356, -84.436, 168.591, 71.27, 3.708]
  MoveL 7996 to (-25.96, 35.46, 116.27) mm, rotated rx -180 ry 0 rz 180 deg; joints [-169.202, 65.356, -84.436, 168.591, 71.27, 3.708]
  Call Extruder(72.39527)
  MoveL 7997 to (-25.65, 35.42, 116.27) mm, rotated rx -180 ry 0 rz 180 deg; joints [-169.199, 65.33, -84.45, 168.585, 71.232, 3.717]
  MoveL 7998 to (-25.65, 35.42, 116.27) mm, rotated rx -180 ry 0 rz 180 deg; joints [-169.199, 65.33, -84.45, 168.585, 71.232, 3.717]
  Call Extruder(72.55409)
  MoveL 7999 to (-25.34, 35.37, 116.27) mm, rotated rx -180 ry 0 rz 180 deg; joints [-169.196, 65.305, -84.463, 168.579, 71.194, 3.726]
  MoveL 8000 to (-25.34, 35.37, 116.27) mm, rotated rx -180 ry 0 rz 180 deg; joints [-169.196, 65.305, -84.463, 168.579, 71.194, 3.726]
  Call Extruder(72.73276)
  MoveL 8001 to (-25, 35.32, 116.27) mm, rotated rx -180 ry 0 rz -180 deg; joints [-169.191, 65.276, -84.478, 168.57, 71.151, 3.737]
  MoveL 8002 to (-25, 35.32, 116.27) mm, rotated rx -180 ry 0 rz -180 deg; joints [-169.191, 65.276, -84.478, 168.57, 71.151, 3.737]
  Call Extruder(72.93120)
  MoveL 8003 to (-24.61, 35.28, 116.27) mm, rotated rx 180 ry 0 rz 180 deg; joints [-169.182, 65.243, -84.495, 168.558, 71.103, 3.75]
  MoveL 8004 to (-24.61, 35.28, 116.27) mm, rotated rx 180 ry 0 rz 180 deg; joints [-169.182, 65.243, -84.495, 168.558, 71.103, 3.75]
  Call Extruder(73.12878)
  MoveL 8005 to (-24.22, 35.23, 116.27) mm, rotated rx -180 ry 0 rz 180 deg; joints [-169.174, 65.211, -84.512, 168.546, 71.056, 3.763]
  MoveL 8006 to (-24.22, 35.23, 116.27) mm, rotated rx -180 ry 0 rz 180 deg; joints [-169.174, 65.211, -84.512, 168.546, 71.056, 3.763]
  Call Extruder(73.32549)
  MoveL 8007 to (-23.84, 35.18, 116.27) mm, rotated rx -180 ry 0 rz -180 deg; joints [-169.166, 65.178, -84.529, 168.534, 71.008, 3.777]
  MoveL 8008 to (-23.84, 35.18, 116.27) mm, rotated rx -180 ry 0 rz -180 deg; joints [-169.166, 65.178, -84.529, 168.534, 71.008, 3.777]
  Call Extruder(73.52132)
  MoveL 8009 to (-23.45, 35.14, 116.27) mm, rotated rx -180 ry 0 rz -180 deg; joints [-169.157, 65.146, -84.545, 168.521, 70.961, 3.79]
  MoveL 8010 to (-23.45, 35.14, 116.27) mm, rotated rx -180 ry 0 rz -180 deg; joints [-169.157, 65.146, -84.545, 168.521, 70.961, 3.79]
  Call Extruder(73.81672)
  MoveL 8011 to (-22.86, 35.09, 116.27) mm, rotated rx -180 ry 0 rz -180 deg; joints [-169.137, 65.097, -84.57, 168.495, 70.889, 3.813]
  MoveL 8012 to (-22.86, 35.09, 116.27) mm, rotated rx -180 ry 0 rz -180 deg; joints [-169.137, 65.097, -84.57, 168.495, 70.889, 3.813]
  Call Extruder(74.11078)
  MoveL 8013 to (-22.27, 35.05, 116.27) mm, rotated rx 180 ry 0 rz 180 deg; joints [-169.117, 65.047, -84.595, 168.468, 70.818, 3.835]
  MoveL 8014 to (-22.27, 35.05, 116.27) mm, rotated rx 180 ry 0 rz 180 deg; joints [-169.117, 65.047, -84.595, 168.468, 70.818, 3.835]
  Call Extruder(74.40351)
  MoveL 8015 to (-21.68, 35, 116.27) mm, rotated rx -180 ry 0 rz -180 deg; joints [-169.096, 64.998, -84.62, 168.442, 70.746, 3.858]
  MoveL 8016 to (-21.68, 35, 116.27) mm, rotated rx -180 ry 0 rz -180 deg; joints [-169.096, 64.998, -84.62, 168.442, 70.746, 3.858]
  Call Extruder(74.97696)
  MoveL 8017 to (-20.52, 34.95, 116.27) mm, rotated rx 180 ry 0 rz 180 deg; joints [-169.042, 64.901, -84.668, 168.374, 70.608, 3.908]
  MoveL 8018 to (-20.52, 34.95, 116.27) mm, rotated rx 180 ry 0 rz 180 deg; joints [-169.042, 64.901, -84.668, 168.374, 70.608, 3.908]
  Call Extruder(75.69093)
  MoveL 8019 to (-19.06, 34.91, 116.27) mm, rotated rx -180 ry 0 rz -180 deg; joints [-168.967, 64.779, -84.727, 168.282, 70.436, 3.973]
  Call Extruder(192.53767)
  MoveL 8020 to (219.06, 34.91, 116.27) mm, rotated rx 180 ry 0 rz 180 deg; joints [-30.588, 53.32, -86.926, 35.364, 118.455, 18.683]
  Call Extruder(192.96623)
  MoveL 8021 to (219.94, 34.93, 116.27) mm, rotated rx -180 ry 0 rz 180 deg; joints [-30.233, 53.408, -86.928, 34.955, 118.497, 18.445]
  MoveL 8022 to (219.94, 34.93, 116.27) mm, rotated rx -180 ry 0 rz 180 deg; joints [-30.233, 53.408, -86.928, 34.955, 118.497, 18.445]
  Call Extruder(193.53967)
  MoveL 8023 to (221.1, 34.97, 116.27) mm, rotated rx -180 ry 0 rz 180 deg; joints [-29.789, 53.526, -86.93, 34.439, 118.542, 18.141]
  MoveL 8024 to (221.1, 34.97, 116.27) mm, rotated rx -180 ry 0 rz 180 deg; joints [-29.789, 53.526, -86.93, 34.439, 118.542, 18.141]
  Call Extruder(193.97399)
  MoveL 8025 to (221.97, 35.02, 116.27) mm, rotated rx -180 ry 0 rz 180 deg; joints [-29.47, 53.615, -86.931, 34.068, 118.567, 17.919]
  MoveL 8026 to (221.97, 35.02, 116.27) mm, rotated rx -180 ry 0 rz 180 deg; joints [-29.47, 53.615, -86.931, 34.068, 118.567, 17.919]
  Call Extruder(194.26805)
  MoveL 8027 to (222.56, 35.07, 116.27) mm, rotated rx -180 ry 0 rz 180 deg; joints [-29.272, 53.676, -86.932, 33.834, 118.578, 17.778]
  MoveL 8028 to (222.56, 35.07, 116.27) mm, rotated rx -180 ry 0 rz 180 deg; joints [-29.272, 53.676, -86.932, 33.834, 118.578, 17.778]
  Call Extruder(194.56344)
  MoveL 8029 to (223.15, 35.11, 116.27) mm, rotated rx -180 ry 0 rz 180 deg; joints [-29.075, 53.738, -86.933, 33.602, 118.588, 17.637]
  MoveL 8030 to (223.15, 35.11, 116.27) mm, rotated rx -180 ry 0 rz 180 deg; joints [-29.075, 53.738, -86.933, 33.602, 118.588, 17.637]
  Call Extruder(194.80967)
  MoveL 8031 to (223.64, 35.16, 116.27) mm, rotated rx -180 ry 0 rz 180 deg; joints [-28.92, 53.789, -86.933, 33.418, 118.592, 17.525]
  MoveL 8032 to (223.64, 35.16, 116.27) mm, rotated rx -180 ry 0 rz 180 deg; joints [-28.92, 53.789, -86.933, 33.418, 118.592, 17.525]
  Call Extruder(195.00638)
  MoveL 8033 to (224.03, 35.21, 116.27) mm, rotated rx -180 ry 0 rz 180 deg; joints [-28.804, 53.83, -86.933, 33.28, 118.593, 17.439]
  MoveL 8034 to (224.03, 35.21, 116.27) mm, rotated rx -180 ry 0 rz 180 deg; joints [-28.804, 53.83, -86.933, 33.28, 118.593, 17.439]
  Call Extruder(195.20395)
  MoveL 8035 to (224.42, 35.25, 116.27) mm, rotated rx 180 ry 0 rz 180 deg; joints [-28.69, 53.871, -86.934, 33.144, 118.593, 17.354]
  MoveL 8036 to (224.42, 35.25, 116.27) mm, rotated rx 180 ry 0 rz 180 deg; joints [-28.69, 53.871, -86.934, 33.144, 118.593, 17.354]
  Call Extruder(195.40240)
  MoveL 8037 to (224.8, 35.3, 116.27) mm, rotated rx -180 ry 0 rz 180 deg; joints [-28.577, 53.912, -86.934, 33.009, 118.592, 17.27]
  MoveL 8038 to (224.8, 35.3, 116.27) mm, rotated rx -180 ry 0 rz 180 deg; joints [-28.577, 53.912, -86.934, 33.009, 118.592, 17.27]
  Call Extruder(195.60171)
  MoveL 8039 to (225.19, 35.34, 116.27) mm, rotated rx -180 ry 0 rz -180 deg; joints [-28.465, 53.953, -86.934, 32.875, 118.591, 17.186]
  MoveL 8040 to (225.19, 35.34, 116.27) mm, rotated rx -180 ry 0 rz -180 deg; joints [-28.465, 53.953, -86.934, 32.875, 118.591, 17.186]
  Call Extruder(195.76053)
  MoveL 8041 to (225.5, 35.39, 116.27) mm, rotated rx -180 ry 0 rz 180 deg; joints [-28.385, 53.987, -86.934, 32.778, 118.586, 17.124]
  MoveL 8042 to (225.5, 35.39, 116.27) mm, rotated rx -180 ry 0 rz 180 deg; joints [-28.385, 53.987, -86.934, 32.778, 118.586, 17.124]
  Call Extruder(195.92007)
  MoveL 8043 to (225.8, 35.44, 116.27) mm, rotated rx -180 ry 0 rz 180 deg; joints [-28.307, 54.02, -86.934, 32.683, 118.582, 17.063]
  MoveL 8044 to (225.8, 35.44, 116.27) mm, rotated rx -180 ry 0 rz 180 deg; joints [-28.307, 54.02, -86.934, 32.683, 118.582, 17.063]
  Call Extruder(196.08035)
  MoveL 8045 to (226.11, 35.49, 116.27) mm, rotated rx -180 ry 0 rz 180 deg; joints [-28.228, 54.053, -86.934, 32.588, 118.577, 17.002]
  MoveL 8046 to (226.11, 35.49, 116.27) mm, rotated rx -180 ry 0 rz 180 deg; joints [-28.228, 54.053, -86.934, 32.588, 118.577, 17.002]
  Call Extruder(196.24135)
  MoveL 8047 to (226.41, 35.54, 116.27) mm, rotated rx 180 ry 0 rz 180 deg; joints [-28.151, 54.086, -86.934, 32.495, 118.571, 16.942]
  MoveL 8048 to (226.41, 35.54, 116.27) mm, rotated rx 180 ry 0 rz 180 deg; joints [-28.151, 54.086, -86.934, 32.495, 118.571, 16.942]
  Call Extruder(196.40308)
  MoveL 8049 to (226.72, 35.59, 116.27) mm, rotated rx -180 ry 0 rz 180 deg; joints [-28.074, 54.119, -86.934, 32.401, 118.566, 16.881]
  MoveL 8050 to (226.72, 35.59, 116.27) mm, rotated rx -180 ry 0 rz 180 deg; joints [-28.074, 54.119, -86.934, 32.401, 118.566, 16.881]
  Call Extruder(196.56554)
  MoveL 8051 to (227.03, 35.64, 116.27) mm, rotated rx -180 ry 0 rz 180 deg; joints [-27.998, 54.152, -86.934, 32.309, 118.56, 16.821]
  MoveL 8052 to (227.03, 35.64, 116.27) mm, rotated rx -180 ry 0 rz 180 deg; joints [-27.998, 54.152, -86.934, 32.309, 118.56, 16.821]
  Call Extruder(196.69947)
  MoveL 8053 to (227.28, 35.68, 116.27) mm, rotated rx -180 ry 0 rz 180 deg; joints [-27.942, 54.18, -86.934, 32.24, 118.552, 16.776]
  MoveL 8054 to (227.28, 35.68, 116.27) mm, rotated rx -180 ry 0 rz 180 deg; joints [-27.942, 54.18, -86.934, 32.24, 118.552, 16.776]
  Call Extruder(196.83401)
  MoveL 8055 to (227.52, 35.73, 116.27) mm, rotated rx 180 ry 0 rz 180 deg; joints [-27.888, 54.207, -86.934, 32.172, 118.545, 16.73]
  MoveL 8056 to (227.52, 35.73, 116.27) mm, rotated rx 180 ry 0 rz 180 deg; joints [-27.888, 54.207, -86.934, 32.172, 118.545, 16.73]
  Call Extruder(196.96915)
  MoveL 8057 to (227.77, 35.78, 116.27) mm, rotated rx 180 ry 0 rz 180 deg; joints [-27.834, 54.235, -86.934, 32.106, 118.537, 16.686]
  MoveL 8058 to (227.77, 35.78, 116.27) mm, rotated rx 180 ry 0 rz 180 deg; joints [-27.834, 54.235, -86.934, 32.106, 118.537, 16.686]
  Call Extruder(197.10491)
  MoveL 8059 to (228.02, 35.83, 116.27) mm, rotated rx 180 ry 0 rz 180 deg; joints [-27.78, 54.262, -86.933, 32.038, 118.529, 16.641]
  MoveL 8060 to (228.02, 35.83, 116.27) mm, rotated rx 180 ry 0 rz 180 deg; joints [-27.78, 54.262, -86.933, 32.038, 118.529, 16.641]
  Call Extruder(197.24128)
  MoveL 8061 to (228.27, 35.88, 116.27) mm, rotated rx 180 ry 0 rz 180 deg; joints [-27.726, 54.29, -86.933, 31.972, 118.521, 16.596]
  MoveL 8062 to (228.27, 35.88, 116.27) mm, rotated rx 180 ry 0 rz 180 deg; joints [-27.726, 54.29, -86.933, 31.972, 118.521, 16.596]
  Call Extruder(197.37826)
  MoveL 8063 to (228.52, 35.93, 116.27) mm, rotated rx -180 ry 0 rz 180 deg; joints [-27.673, 54.317, -86.933, 31.906, 118.513, 16.551]
  MoveL 8064 to (228.52, 35.93, 116.27) mm, rotated rx -180 ry 0 rz 180 deg; joints [-27.673, 54.317, -86.933, 31.906, 118.513, 16.551]
  Call Extruder(197.51585)
  MoveL 8065 to (228.77, 35.98, 116.27) mm, rotated rx -180 ry 0 rz 180 deg; joints [-27.62, 54.345, -86.933, 31.84, 118.504, 16.507]
  MoveL 8066 to (228.77, 35.98, 116.27) mm, rotated rx -180 ry 0 rz 180 deg; joints [-27.62, 54.345, -86.933, 31.84, 118.504, 16.507]
  Call Extruder(197.62957)
  MoveL 8067 to (228.97, 36.03, 116.27) mm, rotated rx 180 ry 0 rz 180 deg; joints [-27.579, 54.367, -86.933, 31.789, 118.496, 16.472]
  MoveL 8068 to (228.97, 36.03, 116.27) mm, rotated rx 180 ry 0 rz 180 deg; joints [-27.579, 54.367, -86.933, 31.789, 118.496, 16.472]
  Call Extruder(197.74374)
